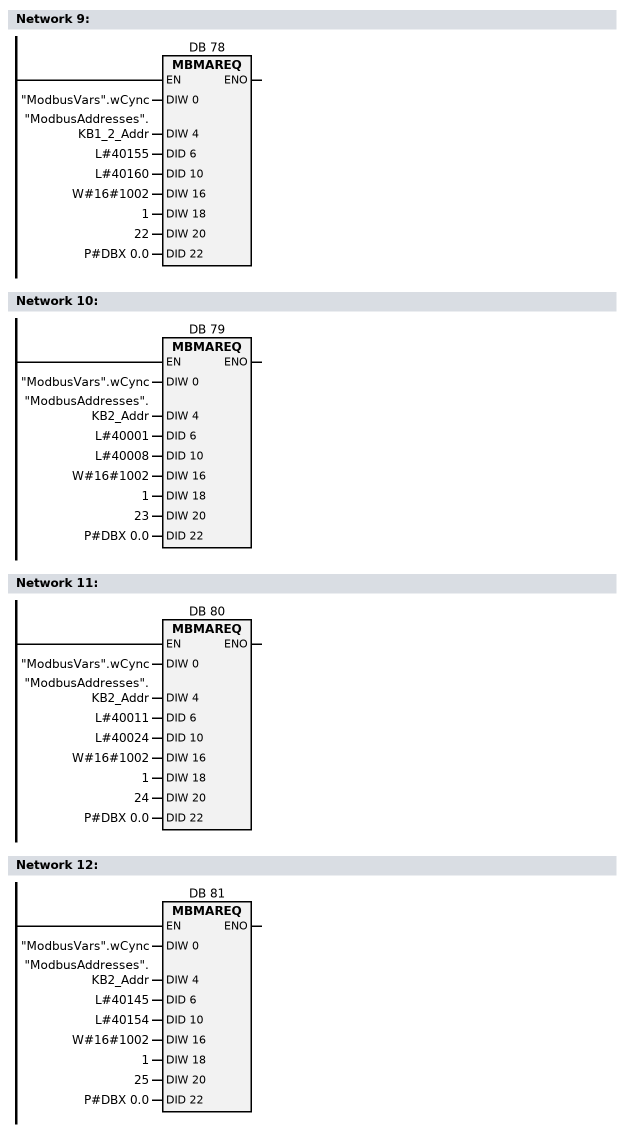
NETWORK
TITLE =
      CALL  "MBMAREQ" , DB 78 (
           DIW 0                    := "ModbusVars".wCync,
           DIW 4                    := "ModbusAddresses".KB1_2_Addr,
           DID 6                    := L#40155,
           DID 10                   := L#40160,
           DIW 16                   := W#16#1002,
           DIW 18                   := 1,
           DIW 20                   := 22,
           DID 22                   := P#DBX 0.0);
      NOP   0;
NETWORK
TITLE =
      CALL  "MBMAREQ" , DB 79 (
           DIW 0                    := "ModbusVars".wCync,
           DIW 4                    := "ModbusAddresses".KB2_Addr,
           DID 6                    := L#40001,
           DID 10                   := L#40008,
           DIW 16                   := W#16#1002,
           DIW 18                   := 1,
           DIW 20                   := 23,
           DID 22                   := P#DBX 0.0);
      NOP   0;
NETWORK
TITLE =
      CALL  "MBMAREQ" , DB 80 (
           DIW 0                    := "ModbusVars".wCync,
           DIW 4                    := "ModbusAddresses".KB2_Addr,
           DID 6                    := L#40011,
           DID 10                   := L#40024,
           DIW 16                   := W#16#1002,
           DIW 18                   := 1,
           DIW 20                   := 24,
           DID 22                   := P#DBX 0.0);
      NOP   0;
NETWORK
TITLE =
      CALL  "MBMAREQ" , DB 81 (
           DIW 0                    := "ModbusVars".wCync,
           DIW 4                    := "ModbusAddresses".KB2_Addr,
           DID 6                    := L#40145,
           DID 10                   := L#40154,
           DIW 16                   := W#16#1002,
           DIW 18                   := 1,
           DIW 20                   := 25,
           DID 22                   := P#DBX 0.0);
      NOP   0;
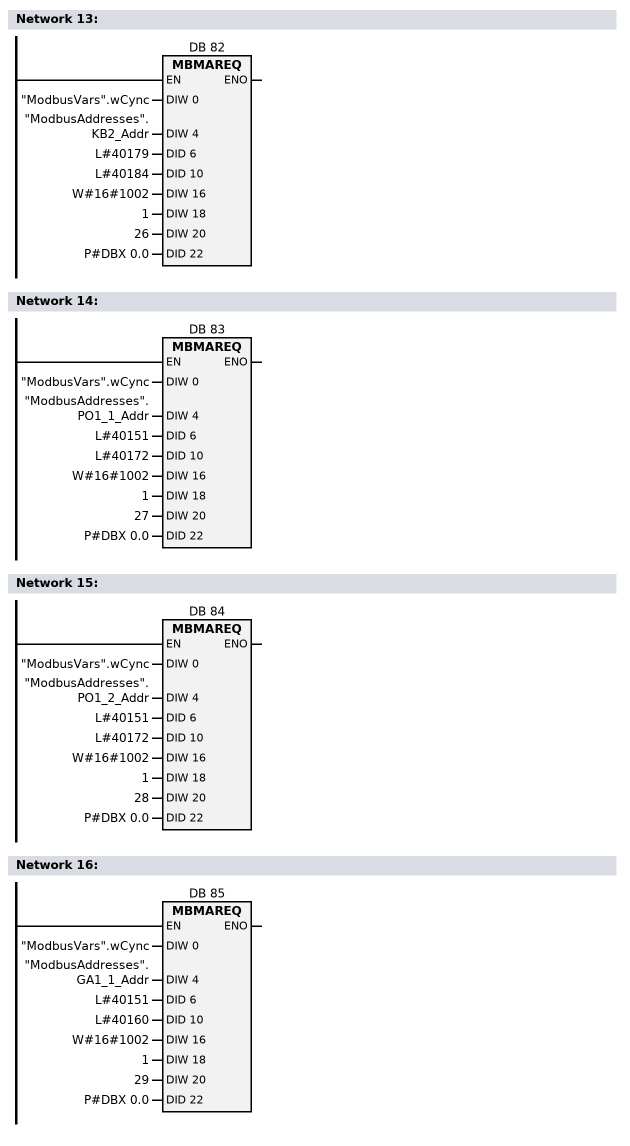
NETWORK
TITLE =
      CALL  "MBMAREQ" , DB 82 (
           DIW 0                    := "ModbusVars".wCync,
           DIW 4                    := "ModbusAddresses".KB2_Addr,
           DID 6                    := L#40179,
           DID 10                   := L#40184,
           DIW 16                   := W#16#1002,
           DIW 18                   := 1,
           DIW 20                   := 26,
           DID 22                   := P#DBX 0.0);
      NOP   0;
NETWORK
TITLE =
      CALL  "MBMAREQ" , DB 83 (
           DIW 0                    := "ModbusVars".wCync,
           DIW 4                    := "ModbusAddresses".PO1_1_Addr,
           DID 6                    := L#40151,
           DID 10                   := L#40172,
           DIW 16                   := W#16#1002,
           DIW 18                   := 1,
           DIW 20                   := 27,
           DID 22                   := P#DBX 0.0);
      NOP   0;
NETWORK
TITLE =
      CALL  "MBMAREQ" , DB 84 (
           DIW 0                    := "ModbusVars".wCync,
           DIW 4                    := "ModbusAddresses".PO1_2_Addr,
           DID 6                    := L#40151,
           DID 10                   := L#40172,
           DIW 16                   := W#16#1002,
           DIW 18                   := 1,
           DIW 20                   := 28,
           DID 22                   := P#DBX 0.0);
      NOP   0;
NETWORK
TITLE =
      CALL  "MBMAREQ" , DB 85 (
           DIW 0                    := "ModbusVars".wCync,
           DIW 4                    := "ModbusAddresses".GA1_1_Addr,
           DID 6                    := L#40151,
           DID 10                   := L#40160,
           DIW 16                   := W#16#1002,
           DIW 18                   := 1,
           DIW 20                   := 29,
           DID 22                   := P#DBX 0.0);
      NOP   0;
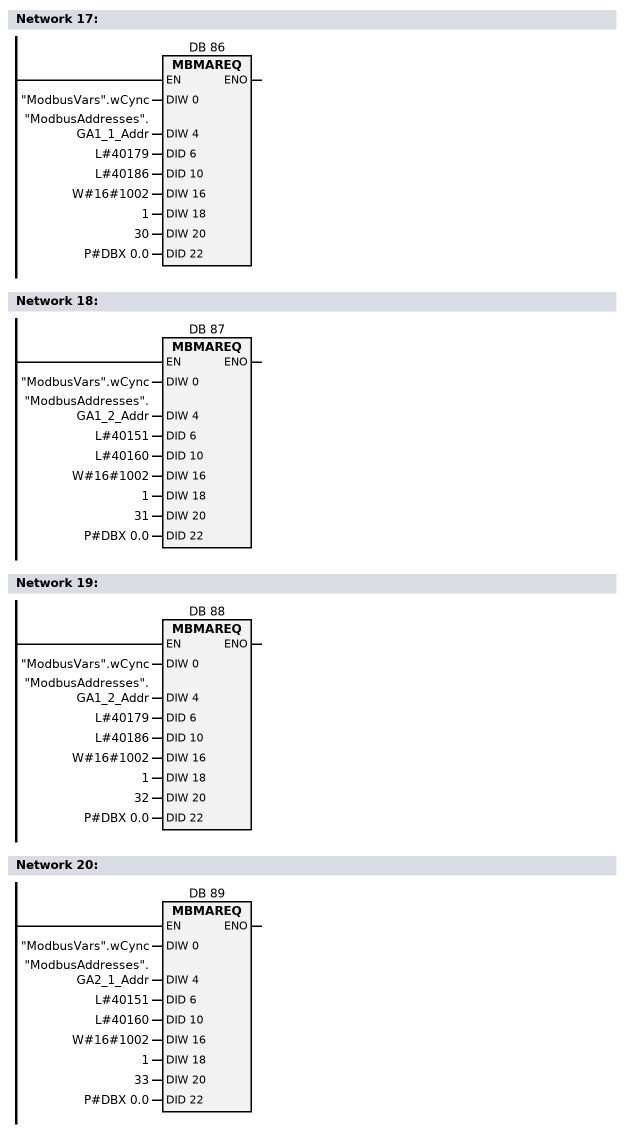
NETWORK
TITLE =
      CALL  "MBMAREQ" , DB 86 (
           DIW 0                    := "ModbusVars".wCync,
           DIW 4                    := "ModbusAddresses".GA1_1_Addr,
           DID 6                    := L#40179,
           DID 10                   := L#40186,
           DIW 16                   := W#16#1002,
           DIW 18                   := 1,
           DIW 20                   := 30,
           DID 22                   := P#DBX 0.0);
      NOP   0;
NETWORK
TITLE =
      CALL  "MBMAREQ" , DB 87 (
           DIW 0                    := "ModbusVars".wCync,
           DIW 4                    := "ModbusAddresses".GA1_2_Addr,
           DID 6                    := L#40151,
           DID 10                   := L#40160,
           DIW 16                   := W#16#1002,
           DIW 18                   := 1,
           DIW 20                   := 31,
           DID 22                   := P#DBX 0.0);
      NOP   0;
NETWORK
TITLE =
      CALL  "MBMAREQ" , DB 88 (
           DIW 0                    := "ModbusVars".wCync,
           DIW 4                    := "ModbusAddresses".GA1_2_Addr,
           DID 6                    := L#40179,
           DID 10                   := L#40186,
           DIW 16                   := W#16#1002,
           DIW 18                   := 1,
           DIW 20                   := 32,
           DID 22                   := P#DBX 0.0);
      NOP   0;
NETWORK
TITLE =
      CALL  "MBMAREQ" , DB 89 (
           DIW 0                    := "ModbusVars".wCync,
           DIW 4                    := "ModbusAddresses".GA2_1_Addr,
           DID 6                    := L#40151,
           DID 10                   := L#40160,
           DIW 16                   := W#16#1002,
           DIW 18                   := 1,
           DIW 20                   := 33,
           DID 22                   := P#DBX 0.0);
      NOP   0;
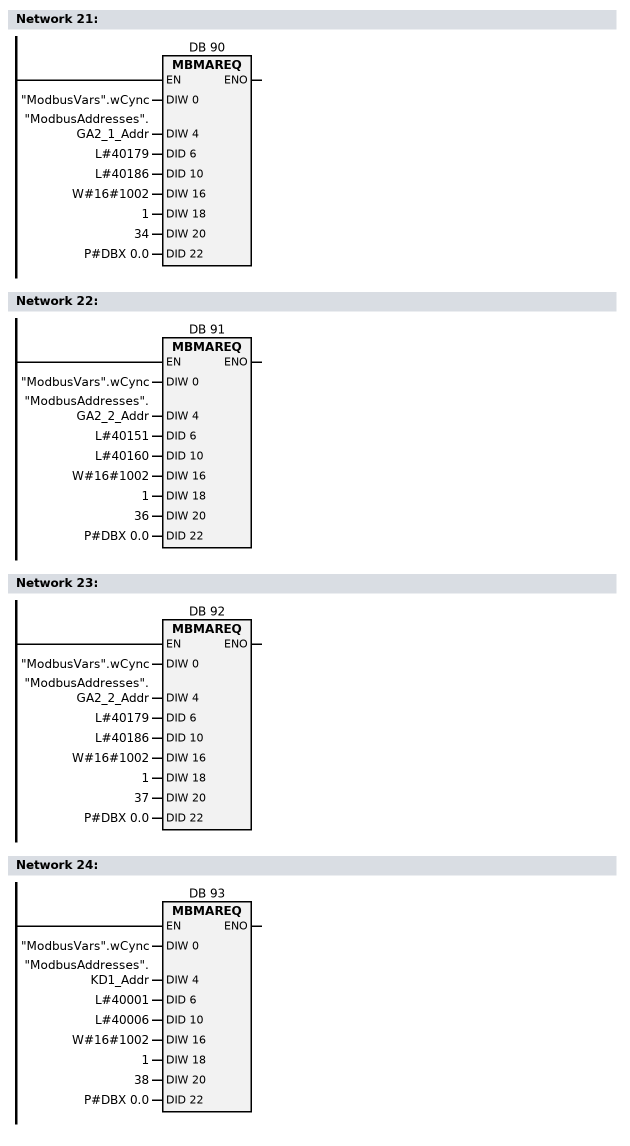
NETWORK
TITLE =
      CALL  "MBMAREQ" , DB 90 (
           DIW 0                    := "ModbusVars".wCync,
           DIW 4                    := "ModbusAddresses".GA2_1_Addr,
           DID 6                    := L#40179,
           DID 10                   := L#40186,
           DIW 16                   := W#16#1002,
           DIW 18                   := 1,
           DIW 20                   := 34,
           DID 22                   := P#DBX 0.0);
      NOP   0;
NETWORK
TITLE =
      CALL  "MBMAREQ" , DB 91 (
           DIW 0                    := "ModbusVars".wCync,
           DIW 4                    := "ModbusAddresses".GA2_2_Addr,
           DID 6                    := L#40151,
           DID 10                   := L#40160,
           DIW 16                   := W#16#1002,
           DIW 18                   := 1,
           DIW 20                   := 36,
           DID 22                   := P#DBX 0.0);
      NOP   0;
NETWORK
TITLE =
      CALL  "MBMAREQ" , DB 92 (
           DIW 0                    := "ModbusVars".wCync,
           DIW 4                    := "ModbusAddresses".GA2_2_Addr,
           DID 6                    := L#40179,
           DID 10                   := L#40186,
           DIW 16                   := W#16#1002,
           DIW 18                   := 1,
           DIW 20                   := 37,
           DID 22                   := P#DBX 0.0);
      NOP   0;
NETWORK
TITLE =
      CALL  "MBMAREQ" , DB 93 (
           DIW 0                    := "ModbusVars".wCync,
           DIW 4                    := "ModbusAddresses".KD1_Addr,
           DID 6                    := L#40001,
           DID 10                   := L#40006,
           DIW 16                   := W#16#1002,
           DIW 18                   := 1,
           DIW 20                   := 38,
           DID 22                   := P#DBX 0.0);
      NOP   0;
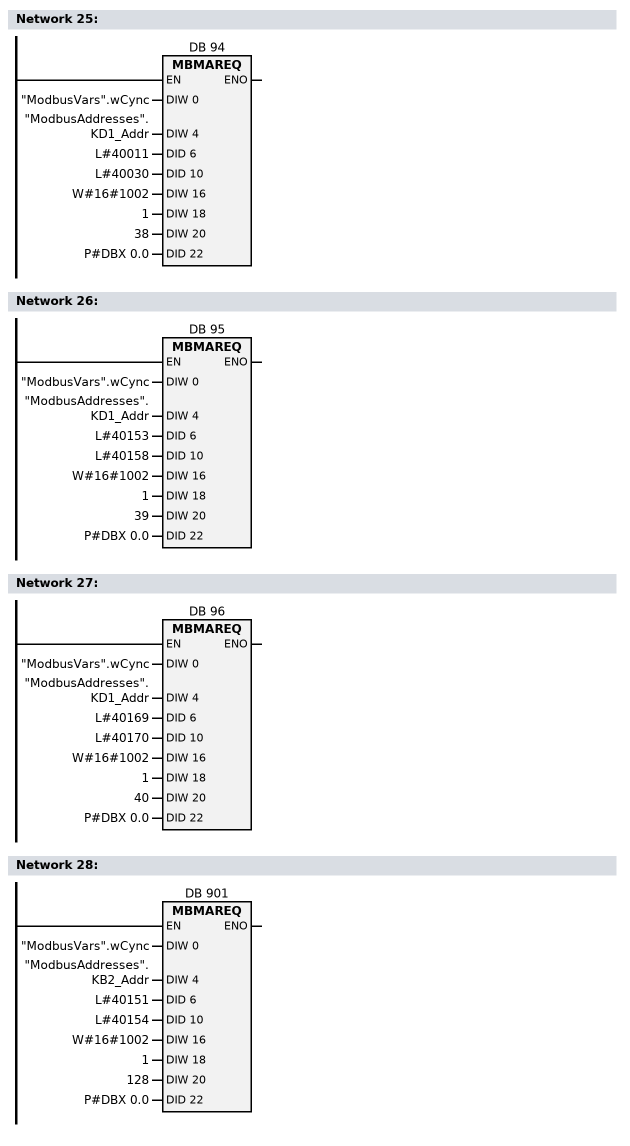
NETWORK
TITLE =
      CALL  "MBMAREQ" , DB 94 (
           DIW 0                    := "ModbusVars".wCync,
           DIW 4                    := "ModbusAddresses".KD1_Addr,
           DID 6                    := L#40011,
           DID 10                   := L#40030,
           DIW 16                   := W#16#1002,
           DIW 18                   := 1,
           DIW 20                   := 38,
           DID 22                   := P#DBX 0.0);
      NOP   0;
NETWORK
TITLE =
      CALL  "MBMAREQ" , DB 95 (
           DIW 0                    := "ModbusVars".wCync,
           DIW 4                    := "ModbusAddresses".KD1_Addr,
           DID 6                    := L#40153,
           DID 10                   := L#40158,
           DIW 16                   := W#16#1002,
           DIW 18                   := 1,
           DIW 20                   := 39,
           DID 22                   := P#DBX 0.0);
      NOP   0;
NETWORK
TITLE =
      CALL  "MBMAREQ" , DB 96 (
           DIW 0                    := "ModbusVars".wCync,
           DIW 4                    := "ModbusAddresses".KD1_Addr,
           DID 6                    := L#40169,
           DID 10                   := L#40170,
           DIW 16                   := W#16#1002,
           DIW 18                   := 1,
           DIW 20                   := 40,
           DID 22                   := P#DBX 0.0);
      NOP   0;
NETWORK
TITLE =
      CALL  "MBMAREQ" , DB 901 (
           DIW 0                    := "ModbusVars".wCync,
           DIW 4                    := "ModbusAddresses".KB2_Addr,
           DID 6                    := L#40151,
           DID 10                   := L#40154,
           DIW 16                   := W#16#1002,
           DIW 18                   := 1,
           DIW 20                   := 128,
           DID 22                   := P#DBX 0.0);
      NOP   0;
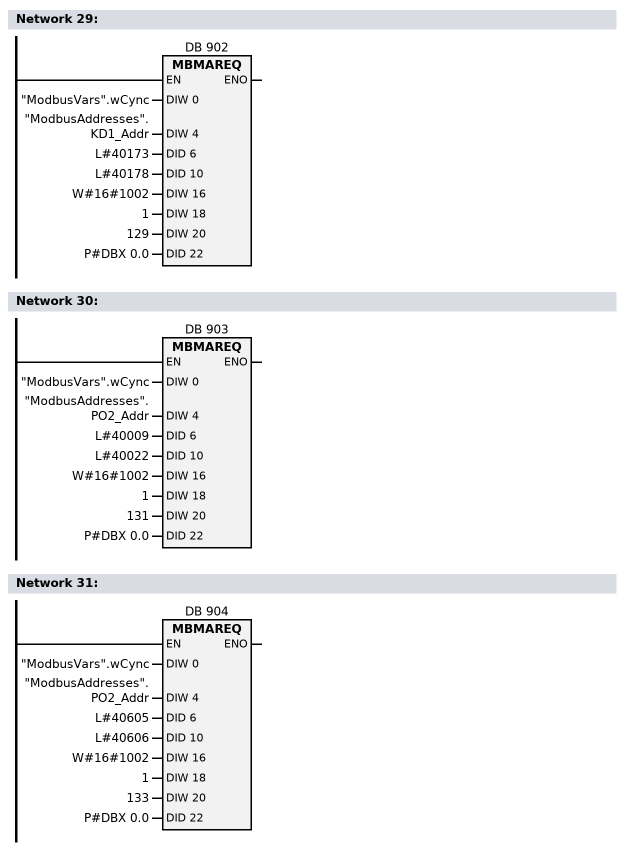
NETWORK
TITLE =
      CALL  "MBMAREQ" , DB 902 (
           DIW 0                    := "ModbusVars".wCync,
           DIW 4                    := "ModbusAddresses".KD1_Addr,
           DID 6                    := L#40173,
           DID 10                   := L#40178,
           DIW 16                   := W#16#1002,
           DIW 18                   := 1,
           DIW 20                   := 129,
           DID 22                   := P#DBX 0.0);
      NOP   0;
NETWORK
TITLE =
      CALL  "MBMAREQ" , DB 903 (
           DIW 0                    := "ModbusVars".wCync,
           DIW 4                    := "ModbusAddresses".PO2_Addr,
           DID 6                    := L#40009,
           DID 10                   := L#40022,
           DIW 16                   := W#16#1002,
           DIW 18                   := 1,
           DIW 20                   := 131,
           DID 22                   := P#DBX 0.0);
      NOP   0;
NETWORK
TITLE =
      CALL  "MBMAREQ" , DB 904 (
           DIW 0                    := "ModbusVars".wCync,
           DIW 4                    := "ModbusAddresses".PO2_Addr,
           DID 6                    := L#40605,
           DID 10                   := L#40606,
           DIW 16                   := W#16#1002,
           DIW 18                   := 1,
           DIW 20                   := 133,
           DID 22                   := P#DBX 0.0);
      NOP   0;
END_FUNCTION_BLOCK

FUNCTION_BLOCK "ModbusCoils"	// FB 16
VERSION : 0.1
BEGIN
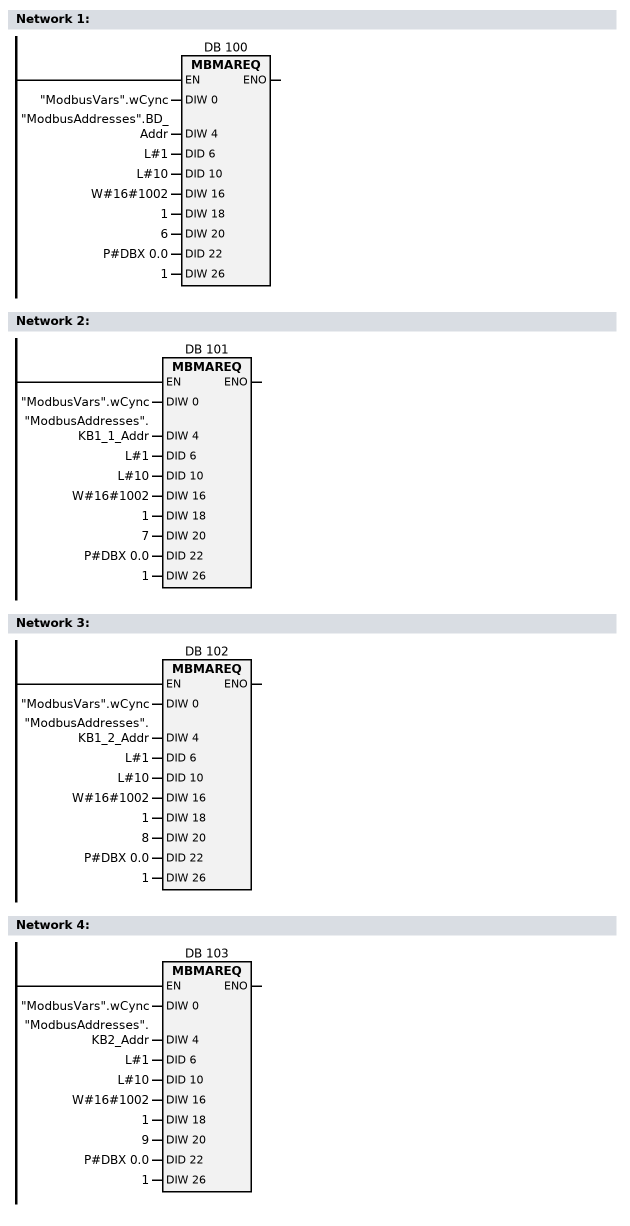
NETWORK
TITLE =
      CALL  "MBMAREQ" , DB 100 (
           DIW 0                    := "ModbusVars".wCync,
           DIW 4                    := "ModbusAddresses".BD_Addr,
           DID 6                    := L#1,
           DID 10                   := L#10,
           DIW 16                   := W#16#1002,
           DIW 18                   := 1,
           DIW 20                   := 6,
           DID 22                   := P#DBX 0.0,
           DIW 26                   := 1);
      NOP   0;
NETWORK
TITLE =
      CALL  "MBMAREQ" , DB 101 (
           DIW 0                    := "ModbusVars".wCync,
           DIW 4                    := "ModbusAddresses".KB1_1_Addr,
           DID 6                    := L#1,
           DID 10                   := L#10,
           DIW 16                   := W#16#1002,
           DIW 18                   := 1,
           DIW 20                   := 7,
           DID 22                   := P#DBX 0.0,
           DIW 26                   := 1);
      NOP   0;
NETWORK
TITLE =
      CALL  "MBMAREQ" , DB 102 (
           DIW 0                    := "ModbusVars".wCync,
           DIW 4                    := "ModbusAddresses".KB1_2_Addr,
           DID 6                    := L#1,
           DID 10                   := L#10,
           DIW 16                   := W#16#1002,
           DIW 18                   := 1,
           DIW 20                   := 8,
           DID 22                   := P#DBX 0.0,
           DIW 26                   := 1);
      NOP   0;
NETWORK
TITLE =
      CALL  "MBMAREQ" , DB 103 (
           DIW 0                    := "ModbusVars".wCync,
           DIW 4                    := "ModbusAddresses".KB2_Addr,
           DID 6                    := L#1,
           DID 10                   := L#10,
           DIW 16                   := W#16#1002,
           DIW 18                   := 1,
           DIW 20                   := 9,
           DID 22                   := P#DBX 0.0,
           DIW 26                   := 1);
      NOP   0;
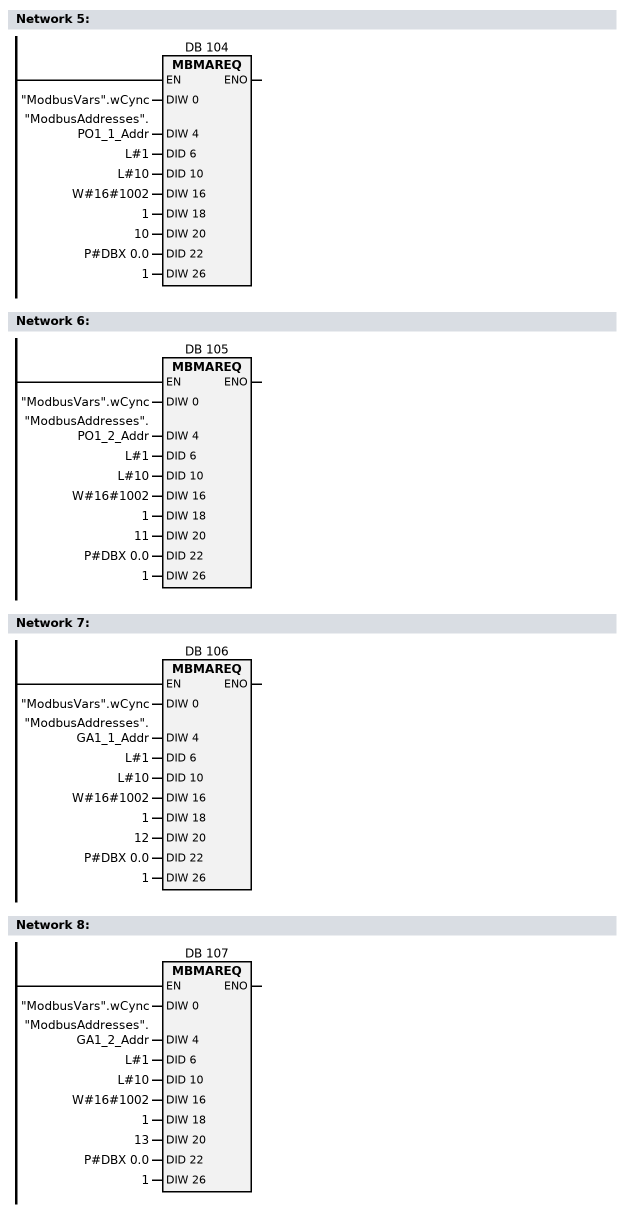
NETWORK
TITLE =
      CALL  "MBMAREQ" , DB 104 (
           DIW 0                    := "ModbusVars".wCync,
           DIW 4                    := "ModbusAddresses".PO1_1_Addr,
           DID 6                    := L#1,
           DID 10                   := L#10,
           DIW 16                   := W#16#1002,
           DIW 18                   := 1,
           DIW 20                   := 10,
           DID 22                   := P#DBX 0.0,
           DIW 26                   := 1);
      NOP   0;
NETWORK
TITLE =
      CALL  "MBMAREQ" , DB 105 (
           DIW 0                    := "ModbusVars".wCync,
           DIW 4                    := "ModbusAddresses".PO1_2_Addr,
           DID 6                    := L#1,
           DID 10                   := L#10,
           DIW 16                   := W#16#1002,
           DIW 18                   := 1,
           DIW 20                   := 11,
           DID 22                   := P#DBX 0.0,
           DIW 26                   := 1);
      NOP   0;
NETWORK
TITLE =
      CALL  "MBMAREQ" , DB 106 (
           DIW 0                    := "ModbusVars".wCync,
           DIW 4                    := "ModbusAddresses".GA1_1_Addr,
           DID 6                    := L#1,
           DID 10                   := L#10,
           DIW 16                   := W#16#1002,
           DIW 18                   := 1,
           DIW 20                   := 12,
           DID 22                   := P#DBX 0.0,
           DIW 26                   := 1);
      NOP   0;
NETWORK
TITLE =
      CALL  "MBMAREQ" , DB 107 (
           DIW 0                    := "ModbusVars".wCync,
           DIW 4                    := "ModbusAddresses".GA1_2_Addr,
           DID 6                    := L#1,
           DID 10                   := L#10,
           DIW 16                   := W#16#1002,
           DIW 18                   := 1,
           DIW 20                   := 13,
           DID 22                   := P#DBX 0.0,
           DIW 26                   := 1);
      NOP   0;
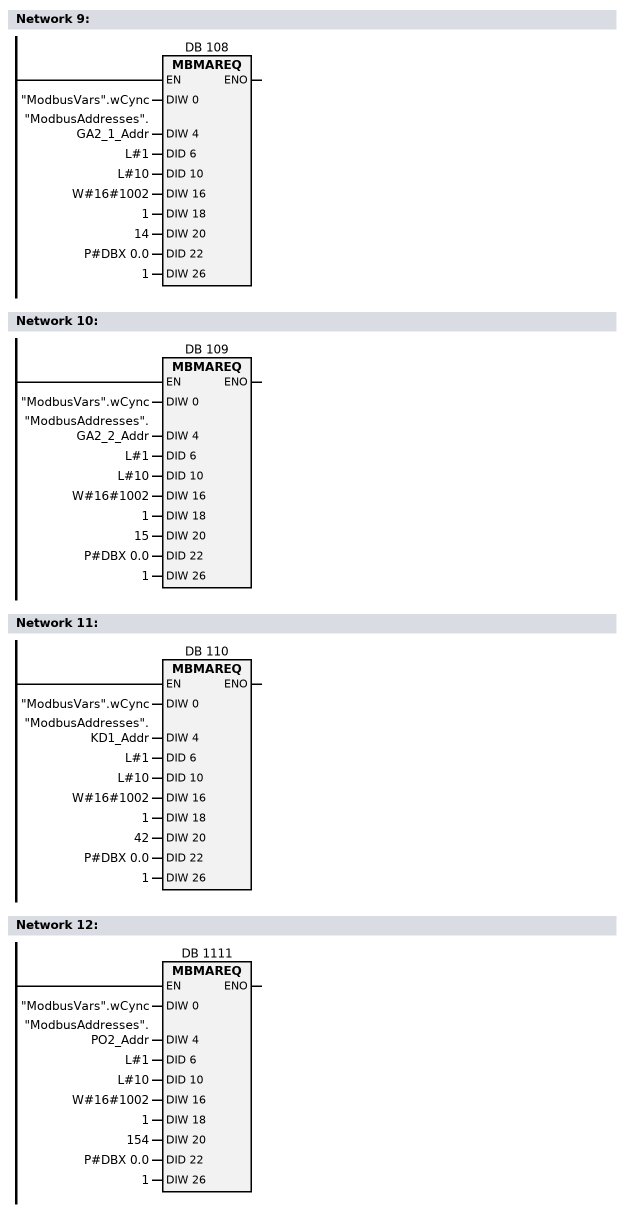
NETWORK
TITLE =
      CALL  "MBMAREQ" , DB 108 (
           DIW 0                    := "ModbusVars".wCync,
           DIW 4                    := "ModbusAddresses".GA2_1_Addr,
           DID 6                    := L#1,
           DID 10                   := L#10,
           DIW 16                   := W#16#1002,
           DIW 18                   := 1,
           DIW 20                   := 14,
           DID 22                   := P#DBX 0.0,
           DIW 26                   := 1);
      NOP   0;
NETWORK
TITLE =
      CALL  "MBMAREQ" , DB 109 (
           DIW 0                    := "ModbusVars".wCync,
           DIW 4                    := "ModbusAddresses".GA2_2_Addr,
           DID 6                    := L#1,
           DID 10                   := L#10,
           DIW 16                   := W#16#1002,
           DIW 18                   := 1,
           DIW 20                   := 15,
           DID 22                   := P#DBX 0.0,
           DIW 26                   := 1);
      NOP   0;
NETWORK
TITLE =
      CALL  "MBMAREQ" , DB 110 (
           DIW 0                    := "ModbusVars".wCync,
           DIW 4                    := "ModbusAddresses".KD1_Addr,
           DID 6                    := L#1,
           DID 10                   := L#10,
           DIW 16                   := W#16#1002,
           DIW 18                   := 1,
           DIW 20                   := 42,
           DID 22                   := P#DBX 0.0,
           DIW 26                   := 1);
      NOP   0;
NETWORK
TITLE =
      CALL  "MBMAREQ" , DB 1111 (
           DIW 0                    := "ModbusVars".wCync,
           DIW 4                    := "ModbusAddresses".PO2_Addr,
           DID 6                    := L#1,
           DID 10                   := L#10,
           DIW 16                   := W#16#1002,
           DIW 18                   := 1,
           DIW 20                   := 154,
           DID 22                   := P#DBX 0.0,
           DIW 26                   := 1);
      NOP   0;
END_FUNCTION_BLOCK

FUNCTION_BLOCK "ModbusOutputs"	// FB 17
VERSION : 0.1
BEGIN
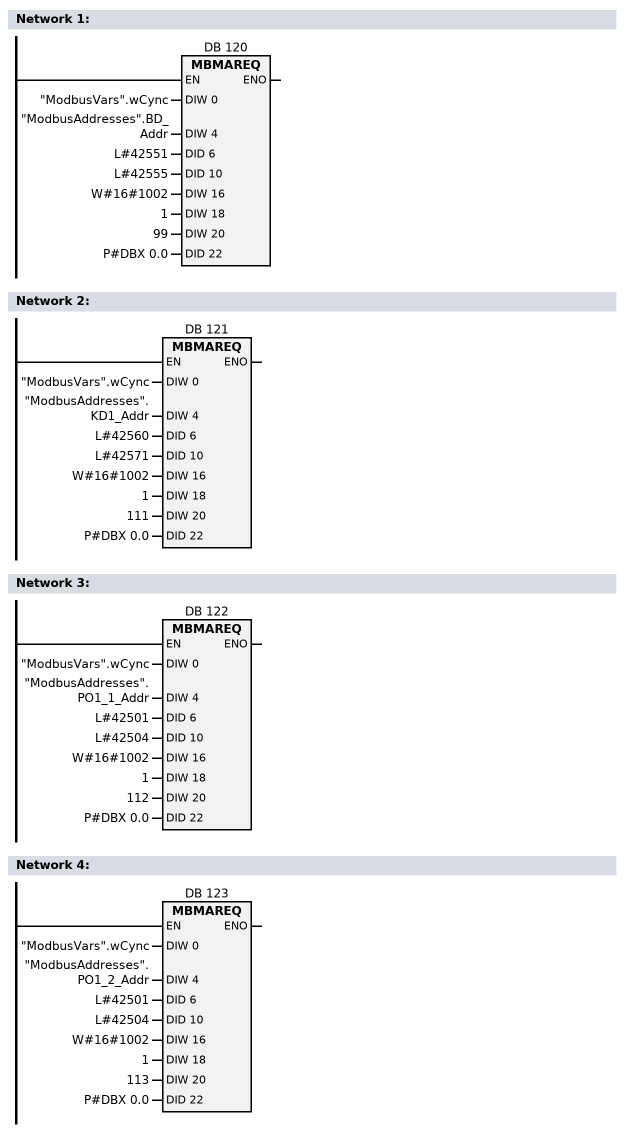
NETWORK
TITLE =
      CALL  "MBMAREQ" , DB 120 (
           DIW 0                    := "ModbusVars".wCync,
           DIW 4                    := "ModbusAddresses".BD_Addr,
           DID 6                    := L#42551,
           DID 10                   := L#42555,
           DIW 16                   := W#16#1002,
           DIW 18                   := 1,
           DIW 20                   := 99,
           DID 22                   := P#DBX 0.0);
      NOP   0;
NETWORK
TITLE =
      CALL  "MBMAREQ" , DB 121 (
           DIW 0                    := "ModbusVars".wCync,
           DIW 4                    := "ModbusAddresses".KD1_Addr,
           DID 6                    := L#42560,
           DID 10                   := L#42571,
           DIW 16                   := W#16#1002,
           DIW 18                   := 1,
           DIW 20                   := 111,
           DID 22                   := P#DBX 0.0);
      NOP   0;
NETWORK
TITLE =
      CALL  "MBMAREQ" , DB 122 (
           DIW 0                    := "ModbusVars".wCync,
           DIW 4                    := "ModbusAddresses".PO1_1_Addr,
           DID 6                    := L#42501,
           DID 10                   := L#42504,
           DIW 16                   := W#16#1002,
           DIW 18                   := 1,
           DIW 20                   := 112,
           DID 22                   := P#DBX 0.0);
      NOP   0;
NETWORK
TITLE =
      CALL  "MBMAREQ" , DB 123 (
           DIW 0                    := "ModbusVars".wCync,
           DIW 4                    := "ModbusAddresses".PO1_2_Addr,
           DID 6                    := L#42501,
           DID 10                   := L#42504,
           DIW 16                   := W#16#1002,
           DIW 18                   := 1,
           DIW 20                   := 113,
           DID 22                   := P#DBX 0.0);
      NOP   0;
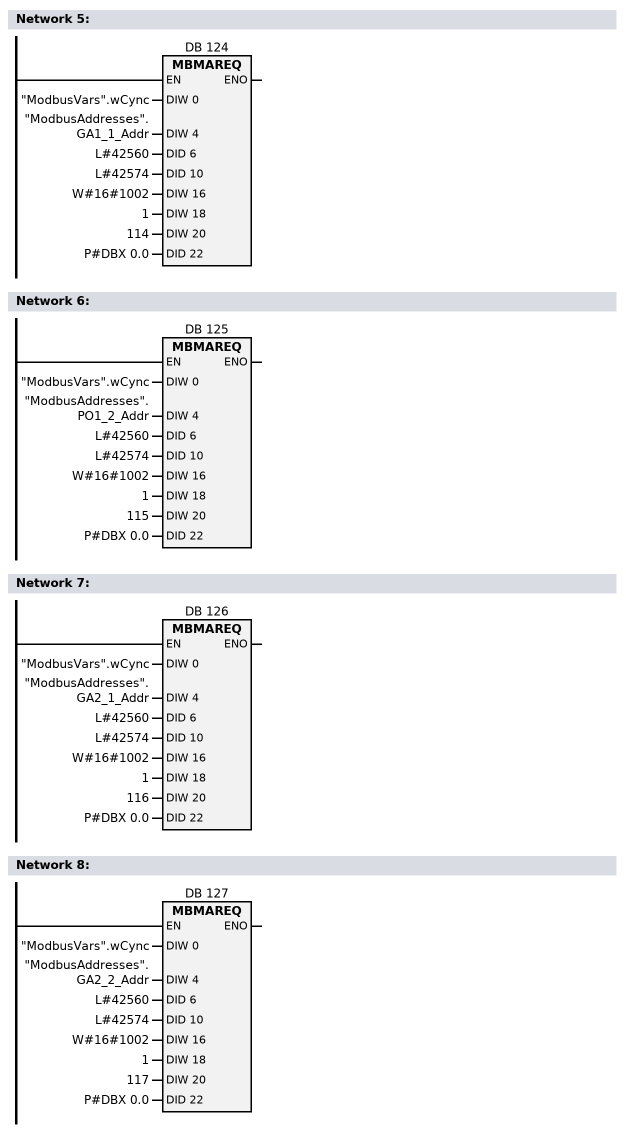
NETWORK
TITLE =
      CALL  "MBMAREQ" , DB 124 (
           DIW 0                    := "ModbusVars".wCync,
           DIW 4                    := "ModbusAddresses".GA1_1_Addr,
           DID 6                    := L#42560,
           DID 10                   := L#42574,
           DIW 16                   := W#16#1002,
           DIW 18                   := 1,
           DIW 20                   := 114,
           DID 22                   := P#DBX 0.0);
      NOP   0;
NETWORK
TITLE =
      CALL  "MBMAREQ" , DB 125 (
           DIW 0                    := "ModbusVars".wCync,
           DIW 4                    := "ModbusAddresses".PO1_2_Addr,
           DID 6                    := L#42560,
           DID 10                   := L#42574,
           DIW 16                   := W#16#1002,
           DIW 18                   := 1,
           DIW 20                   := 115,
           DID 22                   := P#DBX 0.0);
      NOP   0;
NETWORK
TITLE =
      CALL  "MBMAREQ" , DB 126 (
           DIW 0                    := "ModbusVars".wCync,
           DIW 4                    := "ModbusAddresses".GA2_1_Addr,
           DID 6                    := L#42560,
           DID 10                   := L#42574,
           DIW 16                   := W#16#1002,
           DIW 18                   := 1,
           DIW 20                   := 116,
           DID 22                   := P#DBX 0.0);
      NOP   0;
NETWORK
TITLE =
      CALL  "MBMAREQ" , DB 127 (
           DIW 0                    := "ModbusVars".wCync,
           DIW 4                    := "ModbusAddresses".GA2_2_Addr,
           DID 6                    := L#42560,
           DID 10                   := L#42574,
           DIW 16                   := W#16#1002,
           DIW 18                   := 1,
           DIW 20                   := 117,
           DID 22                   := P#DBX 0.0);
      NOP   0;
END_FUNCTION_BLOCK

FUNCTION_BLOCK "BD_GetOutputs"	// FB 18
VERSION : 0.1
BEGIN
NETWORK
TITLE =
      CALL  "fnWordPack" (
           bHigh                    := "BD_OutputBytes_1".arBytes[0],
           bLow                     := "BD_OutputBytes_1".arBytes[1],
           OUT                      := "BD_Outputs_1".DryerMotor);
NETWORK
TITLE =
      CALL  "fnWordPack" (
           bHigh                    := "BD_OutputBytes_1".arBytes[2],
           bLow                     := "BD_OutputBytes_1".arBytes[3],
           OUT                      := "BD_Outputs_1".PDPAlarm);
NETWORK
TITLE =
      CALL  "fnWordPack" (
           bHigh                    := "BD_OutputBytes_1".arBytes[4],
           bLow                     := "BD_OutputBytes_1".arBytes[5],
           OUT                      := "BD_Outputs_1".GeneralShutdown);
NETWORK
TITLE =
      CALL  "fnWordPack" (
           bHigh                    := "BD_OutputBytes_1".arBytes[6],
           bLow                     := "BD_OutputBytes_1".arBytes[7],
           OUT                      := "BD_Outputs_1".GeneralWarning);
NETWORK
TITLE =
      CALL  "fnWordPack" (
           bHigh                    := "BD_OutputBytes_1".arBytes[8],
           bLow                     := "BD_OutputBytes_1".arBytes[9],
           OUT                      := "BD_Outputs_1".LowPressureAlarm);
NETWORK
TITLE =
      CALL  "fnWordPack" (
           bHigh                    := "BD_OutputBytes_2".arBytes[0],
           bLow                     := "BD_OutputBytes_2".arBytes[1],
           OUT                      := "BD_Outputs_2".BlowerContactor);
NETWORK
TITLE =
      CALL  "fnWordPack" (
           bHigh                    := "BD_OutputBytes_2".arBytes[2],
           bLow                     := "BD_OutputBytes_2".arBytes[3],
           OUT                      := "BD_Outputs_2".MainHeaters);
NETWORK
TITLE =
      CALL  "fnWordPack" (
           bHigh                    := "BD_OutputBytes_2".arBytes[4],
           bLow                     := "BD_OutputBytes_2".arBytes[5],
           OUT                      := "BD_Outputs_2".RegulatingHeaters);
NETWORK
TITLE =
      CALL  "fnWordPack" (
           bHigh                    := "BD_OutputBytes_2".arBytes[6],
           bLow                     := "BD_OutputBytes_2".arBytes[7],
           OUT                      := "BD_Outputs_2".ValveV1Opened);
NETWORK
TITLE =
      CALL  "fnWordPack" (
           bHigh                    := "BD_OutputBytes_2".arBytes[8],
           bLow                     := "BD_OutputBytes_2".arBytes[9],
           OUT                      := "BD_Outputs_2".ValveV1Closed);
NETWORK
TITLE =
      CALL  "fnWordPack" (
           bHigh                    := "BD_OutputBytes_2".arBytes[10],
           bLow                     := "BD_OutputBytes_2".arBytes[11],
           OUT                      := "BD_Outputs_2".ValveV2Opened);
NETWORK
TITLE =
      CALL  "fnWordPack" (
           bHigh                    := "BD_OutputBytes_2".arBytes[12],
           bLow                     := "BD_OutputBytes_2".arBytes[13],
           OUT                      := "BD_Outputs_2".ValveV2Closed);
NETWORK
TITLE =
      CALL  "fnWordPack" (
           bHigh                    := "BD_OutputBytes_2".arBytes[14],
           bLow                     := "BD_OutputBytes_2".arBytes[15],
           OUT                      := "BD_Outputs_2".RegValveVesselA);
NETWORK
TITLE =
      CALL  "fnWordPack" (
           bHigh                    := "BD_OutputBytes_2".arBytes[16],
           bLow                     := "BD_OutputBytes_2".arBytes[17],
           OUT                      := "BD_Outputs_2".RegValveVesselB);
NETWORK
TITLE =
      CALL  "fnWordPack" (
           bHigh                    := "BD_OutputBytes_2".arBytes[18],
           bLow                     := "BD_OutputBytes_2".arBytes[19],
           OUT                      := "BD_Outputs_2".CoolingAirValveAOpen);
NETWORK
TITLE =
      CALL  "fnWordPack" (
           bHigh                    := "BD_OutputBytes_2".arBytes[20],
           bLow                     := "BD_OutputBytes_2".arBytes[21],
           OUT                      := "BD_Outputs_2".CoolingAirValveBOpen);
NETWORK
TITLE =
      CALL  "fnWordPack" (
           bHigh                    := "BD_OutputBytes_2".arBytes[22],
           bLow                     := "BD_OutputBytes_2".arBytes[23],
           OUT                      := "BD_Outputs_2".PressureReliefValveA);
NETWORK
TITLE =
      CALL  "fnWordPack" (
           bHigh                    := "BD_OutputBytes_2".arBytes[24],
           bLow                     := "BD_OutputBytes_2".arBytes[25],
           OUT                      := "BD_Outputs_2".PressureReliefValvegB);
END_FUNCTION_BLOCK

FUNCTION_BLOCK "PO1_1_GetOutputs"	// FB 19
VERSION : 0.1
BEGIN
NETWORK
TITLE =
      CALL  "fnBytesToRealTwoComas" (
           bHigh                    := "PO1_1_OutBytes".arBytes[0],
           bLow                     := "PO1_1_OutBytes".arBytes[1],
           OUT                      := "PO1_1_Outputs".EEV1);
NETWORK
TITLE =
      CALL  "fnBytesToRealTwoComas" (
           bHigh                    := "PO1_1_OutBytes".arBytes[2],
           bLow                     := "PO1_1_OutBytes".arBytes[3],
           OUT                      := "PO1_1_Outputs".EEV2);
NETWORK
TITLE =
      CALL  "fnBytesToRealTwoComas" (
           bHigh                    := "PO1_1_OutBytes".arBytes[4],
           bLow                     := "PO1_1_OutBytes".arBytes[5],
           OUT                      := "PO1_1_Outputs".HGBP1);
NETWORK
TITLE =
      CALL  "fnBytesToRealTwoComas" (
           bHigh                    := "PO1_1_OutBytes".arBytes[6],
           bLow                     := "PO1_1_OutBytes".arBytes[7],
           OUT                      := "PO1_1_Outputs".HGBP2);
END_FUNCTION_BLOCK

FUNCTION_BLOCK "PO1_2_GetOutputs"	// FB 20
VERSION : 0.1
BEGIN
NETWORK
TITLE =
      CALL  "fnBytesToRealTwoComas" (
           bHigh                    := "PO1_2_OutBytes".arBytes[0],
           bLow                     := "PO1_2_OutBytes".arBytes[1],
           OUT                      := "PO1_2_Outputs".EEV1);
NETWORK
TITLE =
      CALL  "fnBytesToRealTwoComas" (
           bHigh                    := "PO1_2_OutBytes".arBytes[2],
           bLow                     := "PO1_2_OutBytes".arBytes[3],
           OUT                      := "PO1_2_Outputs".EEV2);
NETWORK
TITLE =
      CALL  "fnBytesToRealTwoComas" (
           bHigh                    := "PO1_2_OutBytes".arBytes[4],
           bLow                     := "PO1_2_OutBytes".arBytes[5],
           OUT                      := "PO1_2_Outputs".HGBP1);
NETWORK
TITLE =
      CALL  "fnBytesToRealTwoComas" (
           bHigh                    := "PO1_2_OutBytes".arBytes[6],
           bLow                     := "PO1_2_OutBytes".arBytes[7],
           OUT                      := "PO1_2_Outputs".HGBP2);
END_FUNCTION_BLOCK

FUNCTION_BLOCK "GA1_1_GetOutputs"	// FB 21
VERSION : 0.1
BEGIN
NETWORK
TITLE =
      CALL  "fnWordPack" (
           bHigh                    := "GA1_1_OutBytes".arBytes[0],
           bLow                     := "GA1_1_OutBytes".arBytes[1],
           OUT                      := "GA1_1_Outputs".InletValveVesselA);
NETWORK
TITLE =
      CALL  "fnWordPack" (
           bHigh                    := "GA1_1_OutBytes".arBytes[2],
           bLow                     := "GA1_1_OutBytes".arBytes[3],
           OUT                      := "GA1_1_Outputs".InletValveVesselB);
NETWORK
TITLE =
      CALL  "fnWordPack" (
           bHigh                    := "GA1_1_OutBytes".arBytes[4],
           bLow                     := "GA1_1_OutBytes".arBytes[5],
           OUT                      := "GA1_1_Outputs".EqualizationValve);
NETWORK
TITLE =
      CALL  "fnWordPack" (
           bHigh                    := "GA1_1_OutBytes".arBytes[6],
           bLow                     := "GA1_1_OutBytes".arBytes[7],
           OUT                      := "GA1_1_Outputs".RegenValveVesselA);
NETWORK
TITLE =
      CALL  "fnWordPack" (
           bHigh                    := "GA1_1_OutBytes".arBytes[8],
           bLow                     := "GA1_1_OutBytes".arBytes[9],
           OUT                      := "GA1_1_Outputs".RegenValveVesselB);
NETWORK
TITLE =
      CALL  "fnWordPack" (
           bHigh                    := "GA1_1_OutBytes".arBytes[10],
           bLow                     := "GA1_1_OutBytes".arBytes[11],
           OUT                      := "GA1_1_Outputs".ProductionValveVesselA);
NETWORK
TITLE =
      CALL  "fnWordPack" (
           bHigh                    := "GA1_1_OutBytes".arBytes[12],
           bLow                     := "GA1_1_OutBytes".arBytes[13],
           OUT                      := "GA1_1_Outputs".ProductionValveVesselB);
NETWORK
TITLE =
      CALL  "fnWordPack" (
           bHigh                    := "GA1_1_OutBytes".arBytes[14],
           bLow                     := "GA1_1_OutBytes".arBytes[15],
           OUT                      := "GA1_1_Outputs".SolenoidValves);
NETWORK
TITLE =
      CALL  "fnWordPack" (
           bHigh                    := "GA1_1_OutBytes".arBytes[16],
           bLow                     := "GA1_1_OutBytes".arBytes[17],
           OUT                      := "GA1_1_Outputs".ConsumerValve);
NETWORK
TITLE =
      CALL  "fnWordPack" (
           bHigh                    := "GA1_1_OutBytes".arBytes[18],
           bLow                     := "GA1_1_OutBytes".arBytes[19],
           OUT                      := "GA1_1_Outputs".InletFlushingValve);
NETWORK
TITLE =
      CALL  "fnWordPack" (
           bHigh                    := "GA1_1_OutBytes".arBytes[20],
           bLow                     := "GA1_1_OutBytes".arBytes[21],
           OUT                      := "GA1_1_Outputs".ExhaustValve);
NETWORK
TITLE =
      CALL  "fnWordPack" (
           bHigh                    := "GA1_1_OutBytes".arBytes[22],
           bLow                     := "GA1_1_OutBytes".arBytes[23],
           OUT                      := "GA1_1_Outputs".Running);
NETWORK
TITLE =
      CALL  "fnWordPack" (
           bHigh                    := "GA1_1_OutBytes".arBytes[24],
           bLow                     := "GA1_1_OutBytes".arBytes[25],
           OUT                      := "GA1_1_Outputs".SecondRunning);
NETWORK
TITLE =
      CALL  "fnWordPack" (
           bHigh                    := "GA1_1_OutBytes".arBytes[26],
           bLow                     := "GA1_1_OutBytes".arBytes[27],
           OUT                      := "GA1_1_Outputs".GeneralWarning);
NETWORK
TITLE =
      CALL  "fnWordPack" (
           bHigh                    := "GA1_1_OutBytes".arBytes[28],
           bLow                     := "GA1_1_OutBytes".arBytes[29],
           OUT                      := "GA1_1_Outputs".GeneralShutdown);
END_FUNCTION_BLOCK

FUNCTION_BLOCK "GA1_2_GetOutputs"	// FB 22
VERSION : 0.1
BEGIN
NETWORK
TITLE =
      CALL  "fnWordPack" (
           bHigh                    := "GA1_2_OutBytes".arBytes[0],
           bLow                     := "GA1_2_OutBytes".arBytes[1],
           OUT                      := "GA1_2_Outputs".InletValveVesselA);
NETWORK
TITLE =
      CALL  "fnWordPack" (
           bHigh                    := "GA1_2_OutBytes".arBytes[2],
           bLow                     := "GA1_2_OutBytes".arBytes[3],
           OUT                      := "GA1_2_Outputs".InletValveVesselB);
NETWORK
TITLE =
      CALL  "fnWordPack" (
           bHigh                    := "GA1_2_OutBytes".arBytes[4],
           bLow                     := "GA1_2_OutBytes".arBytes[5],
           OUT                      := "GA1_2_Outputs".EqualizationValve);
NETWORK
TITLE =
      CALL  "fnWordPack" (
           bHigh                    := "GA1_2_OutBytes".arBytes[6],
           bLow                     := "GA1_2_OutBytes".arBytes[7],
           OUT                      := "GA1_2_Outputs".RegenValveVesselA);
NETWORK
TITLE =
      CALL  "fnWordPack" (
           bHigh                    := "GA1_2_OutBytes".arBytes[8],
           bLow                     := "GA1_2_OutBytes".arBytes[9],
           OUT                      := "GA1_2_Outputs".RegenValveVesselB);
NETWORK
TITLE =
      CALL  "fnWordPack" (
           bHigh                    := "GA1_2_OutBytes".arBytes[10],
           bLow                     := "GA1_2_OutBytes".arBytes[11],
           OUT                      := "GA1_2_Outputs".ProductionValveVesselA);
NETWORK
TITLE =
      CALL  "fnWordPack" (
           bHigh                    := "GA1_2_OutBytes".arBytes[12],
           bLow                     := "GA1_2_OutBytes".arBytes[13],
           OUT                      := "GA1_2_Outputs".ProductionValveVesselB);
NETWORK
TITLE =
      CALL  "fnWordPack" (
           bHigh                    := "GA1_2_OutBytes".arBytes[14],
           bLow                     := "GA1_2_OutBytes".arBytes[15],
           OUT                      := "GA1_2_Outputs".SolenoidValves);
NETWORK
TITLE =
      CALL  "fnWordPack" (
           bHigh                    := "GA1_2_OutBytes".arBytes[16],
           bLow                     := "GA1_2_OutBytes".arBytes[17],
           OUT                      := "GA1_2_Outputs".ConsumerValve);
NETWORK
TITLE =
      CALL  "fnWordPack" (
           bHigh                    := "GA1_2_OutBytes".arBytes[18],
           bLow                     := "GA1_2_OutBytes".arBytes[19],
           OUT                      := "GA1_2_Outputs".InletFlushingValve);
NETWORK
TITLE =
      CALL  "fnWordPack" (
           bHigh                    := "GA1_2_OutBytes".arBytes[20],
           bLow                     := "GA1_2_OutBytes".arBytes[21],
           OUT                      := "GA1_2_Outputs".ExhaustValve);
NETWORK
TITLE =
      CALL  "fnWordPack" (
           bHigh                    := "GA1_2_OutBytes".arBytes[22],
           bLow                     := "GA1_2_OutBytes".arBytes[23],
           OUT                      := "GA1_2_Outputs".Running);
NETWORK
TITLE =
      CALL  "fnWordPack" (
           bHigh                    := "GA1_2_OutBytes".arBytes[24],
           bLow                     := "GA1_2_OutBytes".arBytes[25],
           OUT                      := "GA1_2_Outputs".SecondRunning);
NETWORK
TITLE =
      CALL  "fnWordPack" (
           bHigh                    := "GA1_2_OutBytes".arBytes[26],
           bLow                     := "GA1_2_OutBytes".arBytes[27],
           OUT                      := "GA1_2_Outputs".GeneralWarning);
NETWORK
TITLE =
      CALL  "fnWordPack" (
           bHigh                    := "GA1_2_OutBytes".arBytes[28],
           bLow                     := "GA1_2_OutBytes".arBytes[29],
           OUT                      := "GA1_2_Outputs".GeneralShutdown);
END_FUNCTION_BLOCK

FUNCTION_BLOCK "GA2_1_GetOutputs"	// FB 23
VERSION : 0.1
BEGIN
NETWORK
TITLE =
      CALL  "fnWordPack" (
           bHigh                    := "GA2_1_OutBytes".arBytes[0],
           bLow                     := "GA2_1_OutBytes".arBytes[1],
           OUT                      := "GA2_1_Outputs".InletValveVesselA);
NETWORK
TITLE =
      CALL  "fnWordPack" (
           bHigh                    := "GA2_1_OutBytes".arBytes[2],
           bLow                     := "GA2_1_OutBytes".arBytes[3],
           OUT                      := "GA2_1_Outputs".InletValveVesselB);
NETWORK
TITLE =
      CALL  "fnWordPack" (
           bHigh                    := "GA2_1_OutBytes".arBytes[4],
           bLow                     := "GA2_1_OutBytes".arBytes[5],
           OUT                      := "GA2_1_Outputs".EqualizationValve);
NETWORK
TITLE =
      CALL  "fnWordPack" (
           bHigh                    := "GA2_1_OutBytes".arBytes[6],
           bLow                     := "GA2_1_OutBytes".arBytes[7],
           OUT                      := "GA2_1_Outputs".RegenValveVesselA);
NETWORK
TITLE =
      CALL  "fnWordPack" (
           bHigh                    := "GA2_1_OutBytes".arBytes[8],
           bLow                     := "GA2_1_OutBytes".arBytes[9],
           OUT                      := "GA2_1_Outputs".RegenValveVesselB);
NETWORK
TITLE =
      CALL  "fnWordPack" (
           bHigh                    := "GA2_1_OutBytes".arBytes[10],
           bLow                     := "GA2_1_OutBytes".arBytes[11],
           OUT                      := "GA2_1_Outputs".ProductionValveVesselA);
NETWORK
TITLE =
      CALL  "fnWordPack" (
           bHigh                    := "GA2_1_OutBytes".arBytes[12],
           bLow                     := "GA2_1_OutBytes".arBytes[13],
           OUT                      := "GA2_1_Outputs".ProductionValveVesselB);
NETWORK
TITLE =
      CALL  "fnWordPack" (
           bHigh                    := "GA2_1_OutBytes".arBytes[14],
           bLow                     := "GA2_1_OutBytes".arBytes[15],
           OUT                      := "GA2_1_Outputs".SolenoidValves);
NETWORK
TITLE =
      CALL  "fnWordPack" (
           bHigh                    := "GA2_1_OutBytes".arBytes[16],
           bLow                     := "GA2_1_OutBytes".arBytes[17],
           OUT                      := "GA2_1_Outputs".ConsumerValve);
NETWORK
TITLE =
      CALL  "fnWordPack" (
           bHigh                    := "GA2_1_OutBytes".arBytes[18],
           bLow                     := "GA2_1_OutBytes".arBytes[19],
           OUT                      := "GA2_1_Outputs".InletFlushingValve);
NETWORK
TITLE =
      CALL  "fnWordPack" (
           bHigh                    := "GA2_1_OutBytes".arBytes[20],
           bLow                     := "GA2_1_OutBytes".arBytes[21],
           OUT                      := "GA2_1_Outputs".ExhaustValve);
NETWORK
TITLE =
      CALL  "fnWordPack" (
           bHigh                    := "GA2_1_OutBytes".arBytes[22],
           bLow                     := "GA2_1_OutBytes".arBytes[23],
           OUT                      := "GA2_1_Outputs".Running);
NETWORK
TITLE =
      CALL  "fnWordPack" (
           bHigh                    := "GA2_1_OutBytes".arBytes[24],
           bLow                     := "GA2_1_OutBytes".arBytes[25],
           OUT                      := "GA2_1_Outputs".SecondRunning);
NETWORK
TITLE =
      CALL  "fnWordPack" (
           bHigh                    := "GA2_1_OutBytes".arBytes[26],
           bLow                     := "GA2_1_OutBytes".arBytes[27],
           OUT                      := "GA2_1_Outputs".GeneralWarning);
NETWORK
TITLE =
      CALL  "fnWordPack" (
           bHigh                    := "GA2_1_OutBytes".arBytes[28],
           bLow                     := "GA2_1_OutBytes".arBytes[29],
           OUT                      := "GA2_1_Outputs".GeneralShutdown);
END_FUNCTION_BLOCK

FUNCTION_BLOCK "GA2_2_GetOutputs"	// FB 24
VERSION : 0.1
BEGIN
NETWORK
TITLE =
      CALL  "fnWordPack" (
           bHigh                    := "GA2_2_OutBytes".arBytes[0],
           bLow                     := "GA2_2_OutBytes".arBytes[1],
           OUT                      := "GA2_2_Outputs".InletValveVesselA);
NETWORK
TITLE =
      CALL  "fnWordPack" (
           bHigh                    := "GA2_2_OutBytes".arBytes[2],
           bLow                     := "GA2_2_OutBytes".arBytes[3],
           OUT                      := "GA2_2_Outputs".InletValveVesselB);
NETWORK
TITLE =
      CALL  "fnWordPack" (
           bHigh                    := "GA2_2_OutBytes".arBytes[4],
           bLow                     := "GA2_2_OutBytes".arBytes[5],
           OUT                      := "GA2_2_Outputs".EqualizationValve);
NETWORK
TITLE =
      CALL  "fnWordPack" (
           bHigh                    := "GA2_2_OutBytes".arBytes[6],
           bLow                     := "GA2_2_OutBytes".arBytes[7],
           OUT                      := "GA2_2_Outputs".RegenValveVesselA);
NETWORK
TITLE =
      CALL  "fnWordPack" (
           bHigh                    := "GA2_2_OutBytes".arBytes[8],
           bLow                     := "GA2_2_OutBytes".arBytes[9],
           OUT                      := "GA2_2_Outputs".RegenValveVesselB);
NETWORK
TITLE =
      CALL  "fnWordPack" (
           bHigh                    := "GA2_2_OutBytes".arBytes[10],
           bLow                     := "GA2_2_OutBytes".arBytes[11],
           OUT                      := "GA2_2_Outputs".ProductionValveVesselA);
NETWORK
TITLE =
      CALL  "fnWordPack" (
           bHigh                    := "GA2_2_OutBytes".arBytes[12],
           bLow                     := "GA2_2_OutBytes".arBytes[13],
           OUT                      := "GA2_2_Outputs".ProductionValveVesselB);
NETWORK
TITLE =
      CALL  "fnWordPack" (
           bHigh                    := "GA2_2_OutBytes".arBytes[14],
           bLow                     := "GA2_2_OutBytes".arBytes[15],
           OUT                      := "GA2_2_Outputs".SolenoidValves);
NETWORK
TITLE =
      CALL  "fnWordPack" (
           bHigh                    := "GA2_2_OutBytes".arBytes[16],
           bLow                     := "GA2_2_OutBytes".arBytes[17],
           OUT                      := "GA2_2_Outputs".ConsumerValve);
NETWORK
TITLE =
      CALL  "fnWordPack" (
           bHigh                    := "GA2_2_OutBytes".arBytes[18],
           bLow                     := "GA2_2_OutBytes".arBytes[19],
           OUT                      := "GA2_2_Outputs".InletFlushingValve);
NETWORK
TITLE =
      CALL  "fnWordPack" (
           bHigh                    := "GA2_2_OutBytes".arBytes[20],
           bLow                     := "GA2_2_OutBytes".arBytes[21],
           OUT                      := "GA2_2_Outputs".ExhaustValve);
NETWORK
TITLE =
      CALL  "fnWordPack" (
           bHigh                    := "GA2_2_OutBytes".arBytes[22],
           bLow                     := "GA2_2_OutBytes".arBytes[23],
           OUT                      := "GA2_2_Outputs".Running);
NETWORK
TITLE =
      CALL  "fnWordPack" (
           bHigh                    := "GA2_2_OutBytes".arBytes[24],
           bLow                     := "GA2_2_OutBytes".arBytes[25],
           OUT                      := "GA2_2_Outputs".SecondRunning);
NETWORK
TITLE =
      CALL  "fnWordPack" (
           bHigh                    := "GA2_2_OutBytes".arBytes[26],
           bLow                     := "GA2_2_OutBytes".arBytes[27],
           OUT                      := "GA2_2_Outputs".GeneralWarning);
NETWORK
TITLE =
      CALL  "fnWordPack" (
           bHigh                    := "GA2_2_OutBytes".arBytes[28],
           bLow                     := "GA2_2_OutBytes".arBytes[29],
           OUT                      := "GA2_2_Outputs".GeneralShutdown);
END_FUNCTION_BLOCK

FUNCTION_BLOCK "ModbusStartStop"	// FB 25
VERSION : 0.1
VAR_TEMP
  xAlwaysOn : BOOL ;
END_VAR
BEGIN
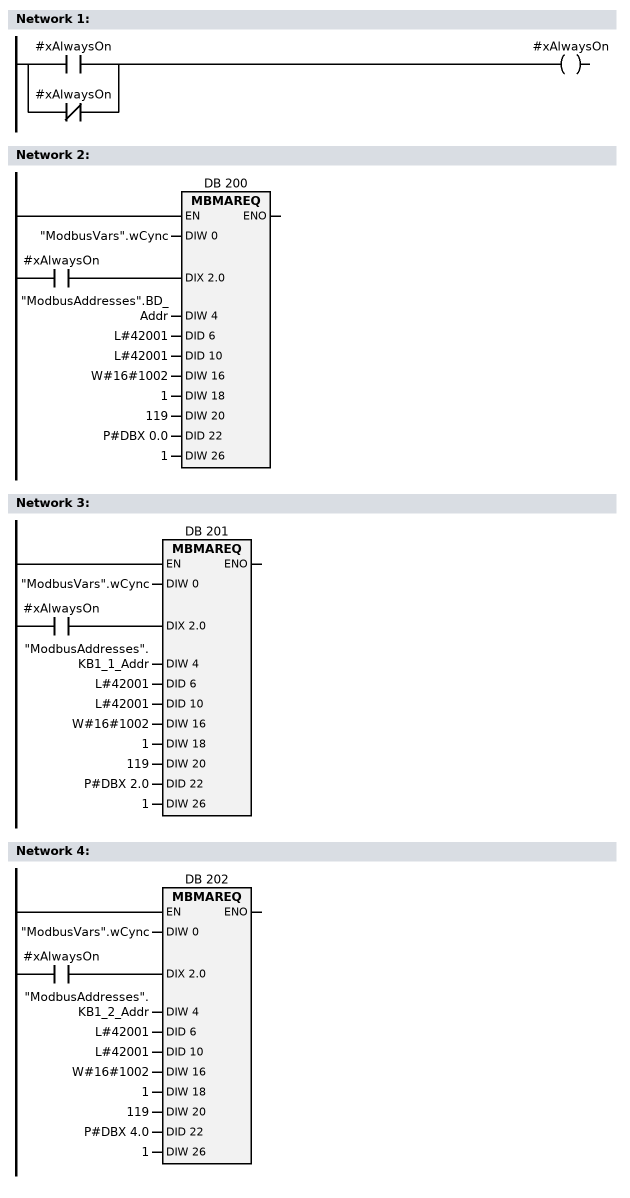
NETWORK
TITLE =
      O     #xAlwaysOn;
      ON    #xAlwaysOn;
      =     #xAlwaysOn;
NETWORK
TITLE =
      A     #xAlwaysOn;
      =     L 1.0;
      BLD   103;
      CALL  "MBMAREQ" , DB 200 (
           DIW 0                    := "ModbusVars".wCync,
           DIX 2.0                  := L 1.0,
           DIW 4                    := "ModbusAddresses".BD_Addr,
           DID 6                    := L#42001,
           DID 10                   := L#42001,
           DIW 16                   := W#16#1002,
           DIW 18                   := 1,
           DIW 20                   := 119,
           DID 22                   := P#DBX 0.0,
           DIW 26                   := 1);
      NOP   0;
NETWORK
TITLE =
      A     #xAlwaysOn;
      =     L 1.0;
      BLD   103;
      CALL  "MBMAREQ" , DB 201 (
           DIW 0                    := "ModbusVars".wCync,
           DIX 2.0                  := L 1.0,
           DIW 4                    := "ModbusAddresses".KB1_1_Addr,
           DID 6                    := L#42001,
           DID 10                   := L#42001,
           DIW 16                   := W#16#1002,
           DIW 18                   := 1,
           DIW 20                   := 119,
           DID 22                   := P#DBX 2.0,
           DIW 26                   := 1);
      NOP   0;
NETWORK
TITLE =
      A     #xAlwaysOn;
      =     L 1.0;
      BLD   103;
      CALL  "MBMAREQ" , DB 202 (
           DIW 0                    := "ModbusVars".wCync,
           DIX 2.0                  := L 1.0,
           DIW 4                    := "ModbusAddresses".KB1_2_Addr,
           DID 6                    := L#42001,
           DID 10                   := L#42001,
           DIW 16                   := W#16#1002,
           DIW 18                   := 1,
           DIW 20                   := 119,
           DID 22                   := P#DBX 4.0,
           DIW 26                   := 1);
      NOP   0;
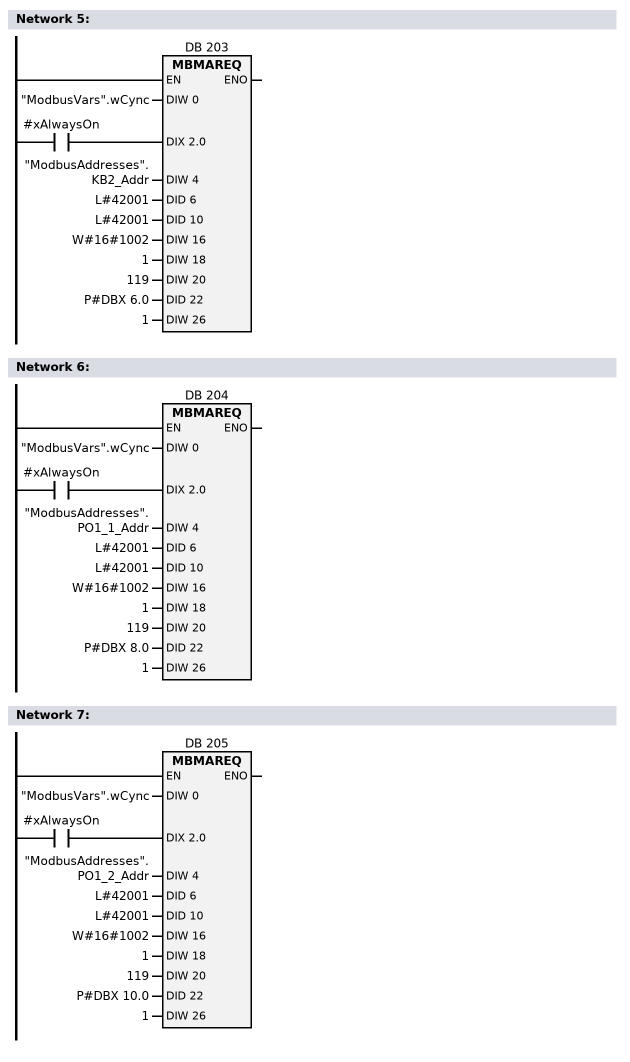
NETWORK
TITLE =
      A     #xAlwaysOn;
      =     L 1.0;
      BLD   103;
      CALL  "MBMAREQ" , DB 203 (
           DIW 0                    := "ModbusVars".wCync,
           DIX 2.0                  := L 1.0,
           DIW 4                    := "ModbusAddresses".KB2_Addr,
           DID 6                    := L#42001,
           DID 10                   := L#42001,
           DIW 16                   := W#16#1002,
           DIW 18                   := 1,
           DIW 20                   := 119,
           DID 22                   := P#DBX 6.0,
           DIW 26                   := 1);
      NOP   0;
NETWORK
TITLE =
      A     #xAlwaysOn;
      =     L 1.0;
      BLD   103;
      CALL  "MBMAREQ" , DB 204 (
           DIW 0                    := "ModbusVars".wCync,
           DIX 2.0                  := L 1.0,
           DIW 4                    := "ModbusAddresses".PO1_1_Addr,
           DID 6                    := L#42001,
           DID 10                   := L#42001,
           DIW 16                   := W#16#1002,
           DIW 18                   := 1,
           DIW 20                   := 119,
           DID 22                   := P#DBX 8.0,
           DIW 26                   := 1);
      NOP   0;
NETWORK
TITLE =
      A     #xAlwaysOn;
      =     L 1.0;
      BLD   103;
      CALL  "MBMAREQ" , DB 205 (
           DIW 0                    := "ModbusVars".wCync,
           DIX 2.0                  := L 1.0,
           DIW 4                    := "ModbusAddresses".PO1_2_Addr,
           DID 6                    := L#42001,
           DID 10                   := L#42001,
           DIW 16                   := W#16#1002,
           DIW 18                   := 1,
           DIW 20                   := 119,
           DID 22                   := P#DBX 10.0,
           DIW 26                   := 1);
      NOP   0;
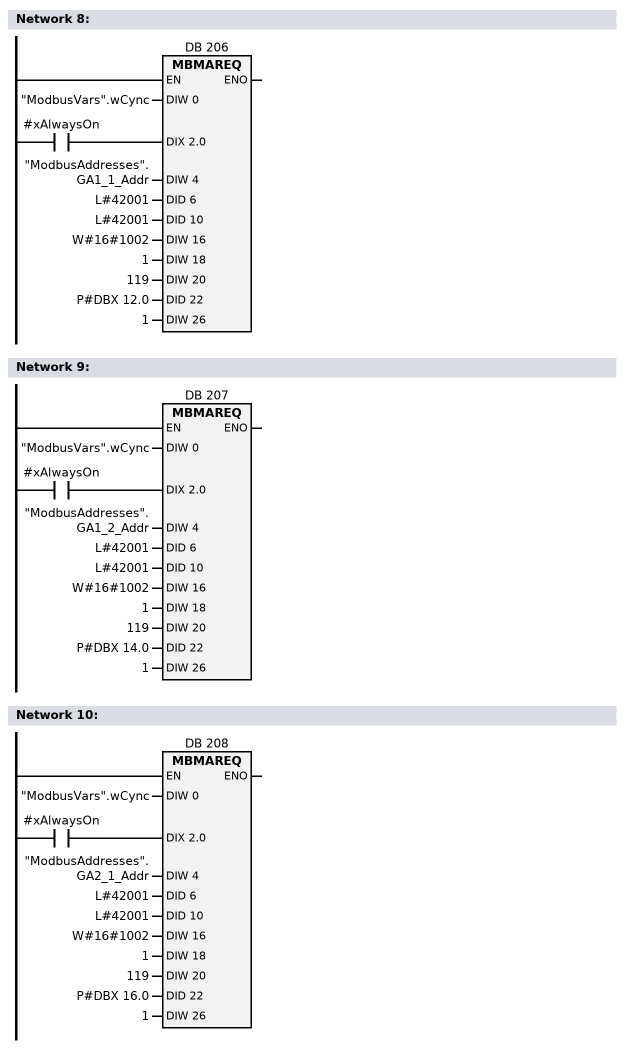
NETWORK
TITLE =
      A     #xAlwaysOn;
      =     L 1.0;
      BLD   103;
      CALL  "MBMAREQ" , DB 206 (
           DIW 0                    := "ModbusVars".wCync,
           DIX 2.0                  := L 1.0,
           DIW 4                    := "ModbusAddresses".GA1_1_Addr,
           DID 6                    := L#42001,
           DID 10                   := L#42001,
           DIW 16                   := W#16#1002,
           DIW 18                   := 1,
           DIW 20                   := 119,
           DID 22                   := P#DBX 12.0,
           DIW 26                   := 1);
      NOP   0;
NETWORK
TITLE =
      A     #xAlwaysOn;
      =     L 1.0;
      BLD   103;
      CALL  "MBMAREQ" , DB 207 (
           DIW 0                    := "ModbusVars".wCync,
           DIX 2.0                  := L 1.0,
           DIW 4                    := "ModbusAddresses".GA1_2_Addr,
           DID 6                    := L#42001,
           DID 10                   := L#42001,
           DIW 16                   := W#16#1002,
           DIW 18                   := 1,
           DIW 20                   := 119,
           DID 22                   := P#DBX 14.0,
           DIW 26                   := 1);
      NOP   0;
NETWORK
TITLE =
      A     #xAlwaysOn;
      =     L 1.0;
      BLD   103;
      CALL  "MBMAREQ" , DB 208 (
           DIW 0                    := "ModbusVars".wCync,
           DIX 2.0                  := L 1.0,
           DIW 4                    := "ModbusAddresses".GA2_1_Addr,
           DID 6                    := L#42001,
           DID 10                   := L#42001,
           DIW 16                   := W#16#1002,
           DIW 18                   := 1,
           DIW 20                   := 119,
           DID 22                   := P#DBX 16.0,
           DIW 26                   := 1);
      NOP   0;
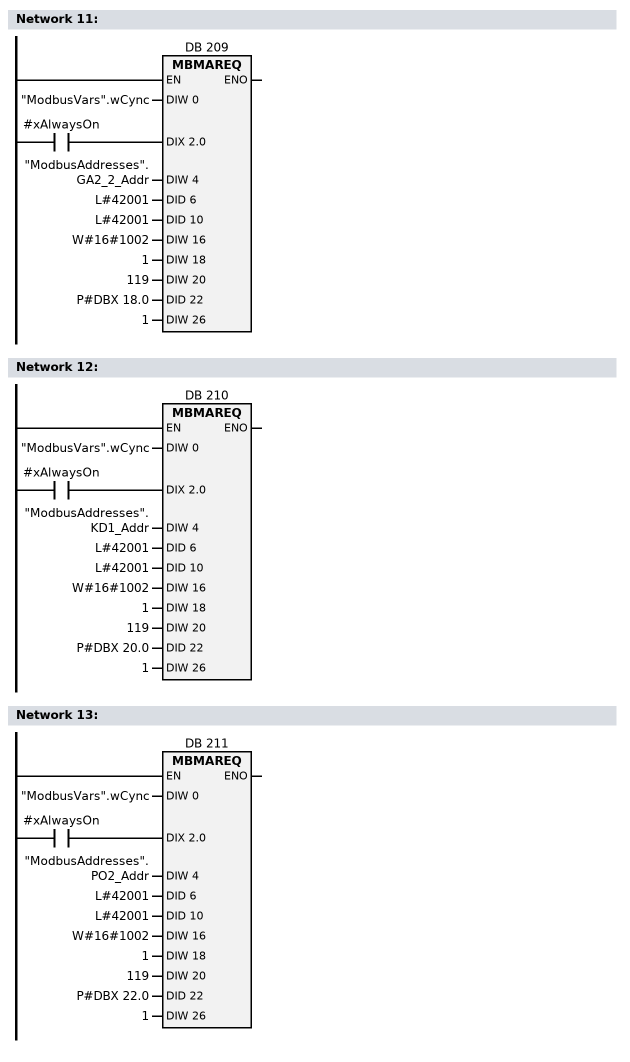
NETWORK
TITLE =
      A     #xAlwaysOn;
      =     L 1.0;
      BLD   103;
      CALL  "MBMAREQ" , DB 209 (
           DIW 0                    := "ModbusVars".wCync,
           DIX 2.0                  := L 1.0,
           DIW 4                    := "ModbusAddresses".GA2_2_Addr,
           DID 6                    := L#42001,
           DID 10                   := L#42001,
           DIW 16                   := W#16#1002,
           DIW 18                   := 1,
           DIW 20                   := 119,
           DID 22                   := P#DBX 18.0,
           DIW 26                   := 1);
      NOP   0;
NETWORK
TITLE =
      A     #xAlwaysOn;
      =     L 1.0;
      BLD   103;
      CALL  "MBMAREQ" , DB 210 (
           DIW 0                    := "ModbusVars".wCync,
           DIX 2.0                  := L 1.0,
           DIW 4                    := "ModbusAddresses".KD1_Addr,
           DID 6                    := L#42001,
           DID 10                   := L#42001,
           DIW 16                   := W#16#1002,
           DIW 18                   := 1,
           DIW 20                   := 119,
           DID 22                   := P#DBX 20.0,
           DIW 26                   := 1);
      NOP   0;
NETWORK
TITLE =
      A     #xAlwaysOn;
      =     L 1.0;
      BLD   103;
      CALL  "MBMAREQ" , DB 211 (
           DIW 0                    := "ModbusVars".wCync,
           DIX 2.0                  := L 1.0,
           DIW 4                    := "ModbusAddresses".PO2_Addr,
           DID 6                    := L#42001,
           DID 10                   := L#42001,
           DIW 16                   := W#16#1002,
           DIW 18                   := 1,
           DIW 20                   := 119,
           DID 22                   := P#DBX 22.0,
           DIW 26                   := 1);
      NOP   0;
END_FUNCTION_BLOCK

FUNCTION_BLOCK "GetStartStopBytes"	// FB 26
VERSION : 0.1
BEGIN
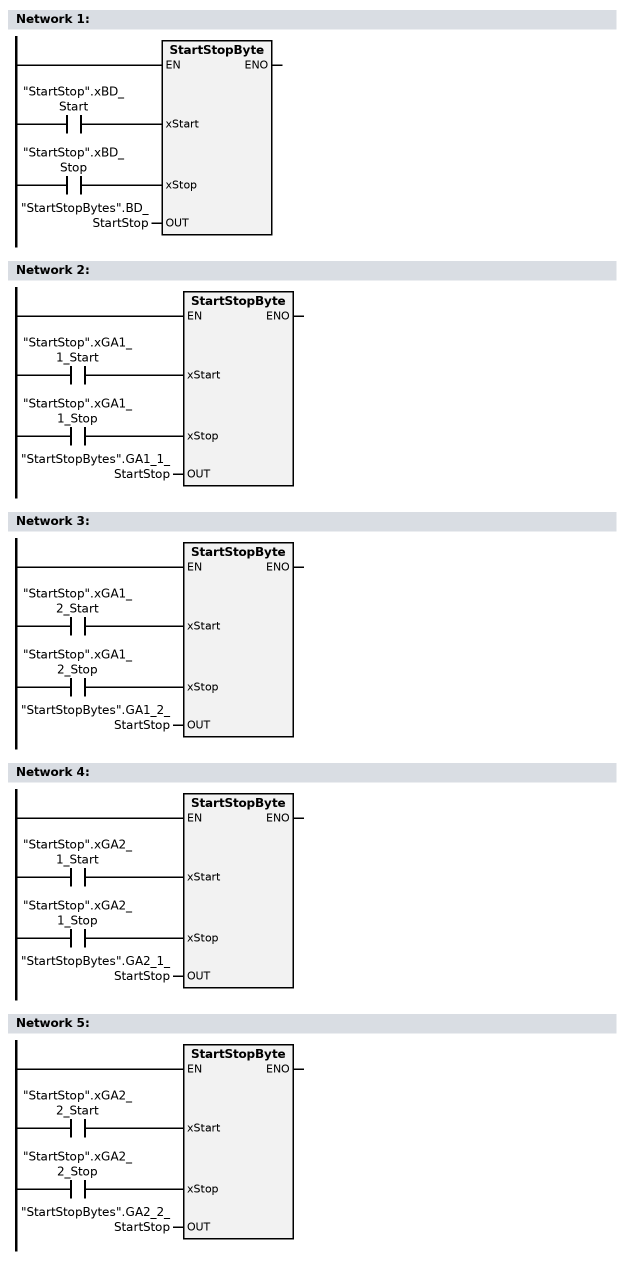
NETWORK
TITLE =
      A     "StartStop".xBD_Start;
      =     L 0.0;
      BLD   103;
      A     "StartStop".xBD_Stop;
      =     L 0.1;
      BLD   103;
      CALL  "StartStopByte" (
           xStart                   := L 0.0,
           xStop                    := L 0.1,
           OUT                      := "StartStopBytes".BD_StartStop);
      NOP   0;
NETWORK
TITLE =
      A     "StartStop".xGA1_1_Start;
      =     L 0.0;
      BLD   103;
      A     "StartStop".xGA1_1_Stop;
      =     L 0.1;
      BLD   103;
      CALL  "StartStopByte" (
           xStart                   := L 0.0,
           xStop                    := L 0.1,
           OUT                      := "StartStopBytes".GA1_1_StartStop);
      NOP   0;
NETWORK
TITLE =
      A     "StartStop".xGA1_2_Start;
      =     L 0.0;
      BLD   103;
      A     "StartStop".xGA1_2_Stop;
      =     L 0.1;
      BLD   103;
      CALL  "StartStopByte" (
           xStart                   := L 0.0,
           xStop                    := L 0.1,
           OUT                      := "StartStopBytes".GA1_2_StartStop);
      NOP   0;
NETWORK
TITLE =
      A     "StartStop".xGA2_1_Start;
      =     L 0.0;
      BLD   103;
      A     "StartStop".xGA2_1_Stop;
      =     L 0.1;
      BLD   103;
      CALL  "StartStopByte" (
           xStart                   := L 0.0,
           xStop                    := L 0.1,
           OUT                      := "StartStopBytes".GA2_1_StartStop);
      NOP   0;
NETWORK
TITLE =
      A     "StartStop".xGA2_2_Start;
      =     L 0.0;
      BLD   103;
      A     "StartStop".xGA2_2_Stop;
      =     L 0.1;
      BLD   103;
      CALL  "StartStopByte" (
           xStart                   := L 0.0,
           xStop                    := L 0.1,
           OUT                      := "StartStopBytes".GA2_2_StartStop);
      NOP   0;
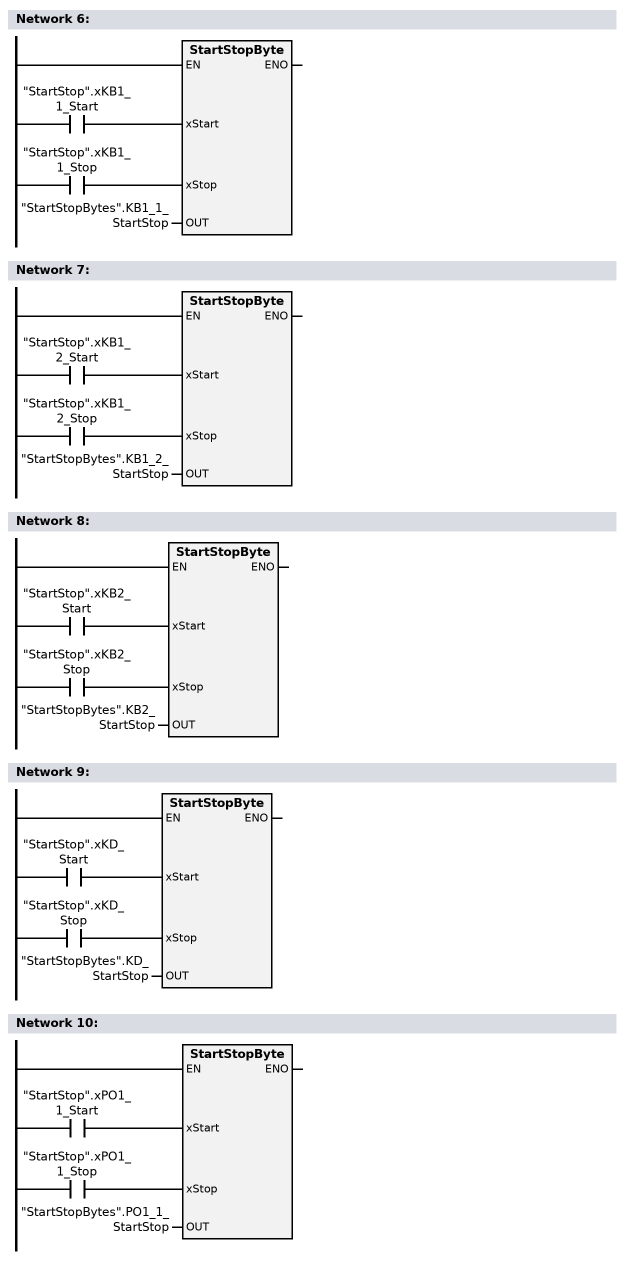
NETWORK
TITLE =
      A     "StartStop".xKB1_1_Start;
      =     L 0.0;
      BLD   103;
      A     "StartStop".xKB1_1_Stop;
      =     L 0.1;
      BLD   103;
      CALL  "StartStopByte" (
           xStart                   := L 0.0,
           xStop                    := L 0.1,
           OUT                      := "StartStopBytes".KB1_1_StartStop);
      NOP   0;
NETWORK
TITLE =
      A     "StartStop".xKB1_2_Start;
      =     L 0.0;
      BLD   103;
      A     "StartStop".xKB1_2_Stop;
      =     L 0.1;
      BLD   103;
      CALL  "StartStopByte" (
           xStart                   := L 0.0,
           xStop                    := L 0.1,
           OUT                      := "StartStopBytes".KB1_2_StartStop);
      NOP   0;
NETWORK
TITLE =
      A     "StartStop".xKB2_Start;
      =     L 0.0;
      BLD   103;
      A     "StartStop".xKB2_Stop;
      =     L 0.1;
      BLD   103;
      CALL  "StartStopByte" (
           xStart                   := L 0.0,
           xStop                    := L 0.1,
           OUT                      := "StartStopBytes".KB2_StartStop);
      NOP   0;
NETWORK
TITLE =
      A     "StartStop".xKD_Start;
      =     L 0.0;
      BLD   103;
      A     "StartStop".xKD_Stop;
      =     L 0.1;
      BLD   103;
      CALL  "StartStopByte" (
           xStart                   := L 0.0,
           xStop                    := L 0.1,
           OUT                      := "StartStopBytes".KD_StartStop);
      NOP   0;
NETWORK
TITLE =
      A     "StartStop".xPO1_1_Start;
      =     L 0.0;
      BLD   103;
      A     "StartStop".xPO1_1_Stop;
      =     L 0.1;
      BLD   103;
      CALL  "StartStopByte" (
           xStart                   := L 0.0,
           xStop                    := L 0.1,
           OUT                      := "StartStopBytes".PO1_1_StartStop);
      NOP   0;
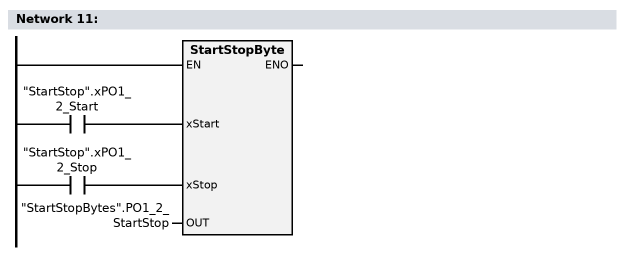
NETWORK
TITLE =
      A     "StartStop".xPO1_2_Start;
      =     L 0.0;
      BLD   103;
      A     "StartStop".xPO1_2_Stop;
      =     L 0.1;
      BLD   103;
      CALL  "StartStopByte" (
           xStart                   := L 0.0,
           xStop                    := L 0.1,
           OUT                      := "StartStopBytes".PO1_2_StartStop);
      NOP   0;
END_FUNCTION_BLOCK

FUNCTION_BLOCK "GetAll"	// FB 27
VERSION : 0.1
BEGIN
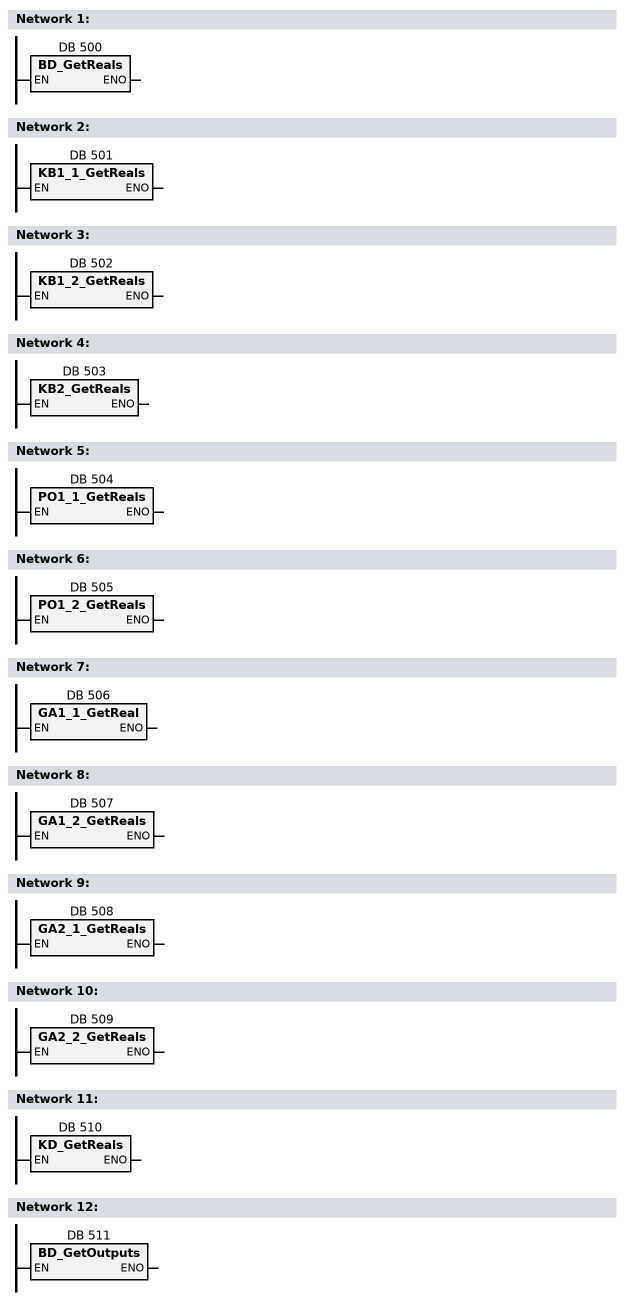
NETWORK
TITLE =
      CALL  "BD_GetReals" , DB 500;
      NOP   0;
NETWORK
TITLE =
      CALL  "KB1_1_GetReals" , DB 501;
      NOP   0;
NETWORK
TITLE =
      CALL  "KB1_2_GetReals" , DB 502;
      NOP   0;
NETWORK
TITLE =
      CALL  "KB2_GetReals" , DB 503;
      NOP   0;
NETWORK
TITLE =
      CALL  "PO1_1_GetReals" , DB 504;
      NOP   0;
NETWORK
TITLE =
      CALL  "PO1_2_GetReals" , DB 505;
      NOP   0;
NETWORK
TITLE =
      CALL  "GA1_1_GetReal" , DB 506;
      NOP   0;
NETWORK
TITLE =
      CALL  "GA1_2_GetReals" , DB 507;
      NOP   0;
NETWORK
TITLE =
      CALL  "GA2_1_GetReals" , DB 508;
      NOP   0;
NETWORK
TITLE =
      CALL  "GA2_2_GetReals" , DB 509;
      NOP   0;
NETWORK
TITLE =
      CALL  "KD_GetReals" , DB 510;
      NOP   0;
NETWORK
TITLE =
      CALL  "BD_GetOutputs" , DB 511;
      NOP   0;
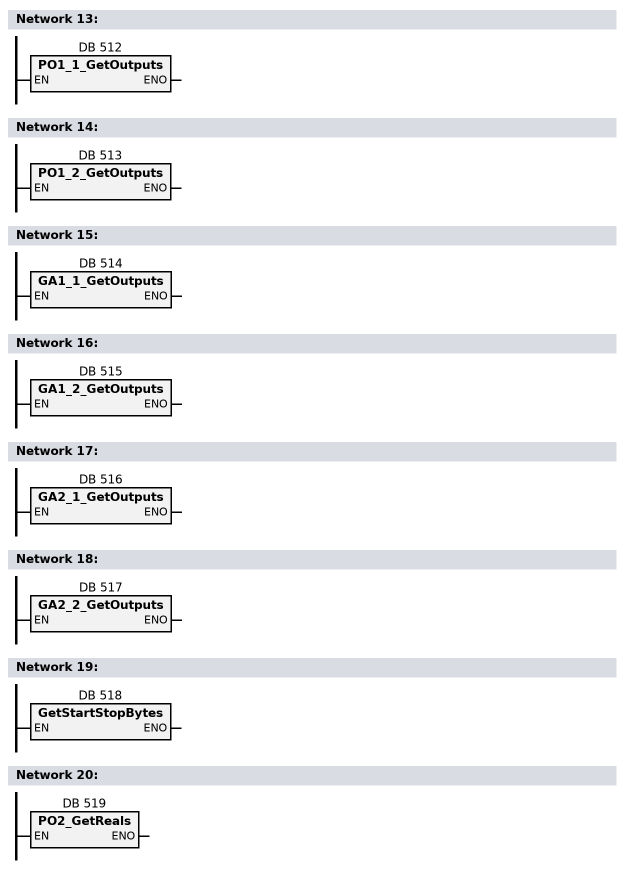
NETWORK
TITLE =
      CALL  "PO1_1_GetOutputs" , DB 512;
      NOP   0;
NETWORK
TITLE =
      CALL  "PO1_2_GetOutputs" , DB 513;
      NOP   0;
NETWORK
TITLE =
      CALL  "GA1_1_GetOutputs" , DB 514;
      NOP   0;
NETWORK
TITLE =
      CALL  "GA1_2_GetOutputs" , DB 515;
      NOP   0;
NETWORK
TITLE =
      CALL  "GA2_1_GetOutputs" , DB 516;
      NOP   0;
NETWORK
TITLE =
      CALL  "GA2_2_GetOutputs" , DB 517;
      NOP   0;
NETWORK
TITLE =
      CALL  "GetStartStopBytes" , DB 518;
      NOP   0;
NETWORK
TITLE =
      CALL  "PO2_GetReals" , DB 519;
      NOP   0;
END_FUNCTION_BLOCK

FUNCTION_BLOCK "ModbusAll"	// FB 28
VERSION : 0.1
BEGIN
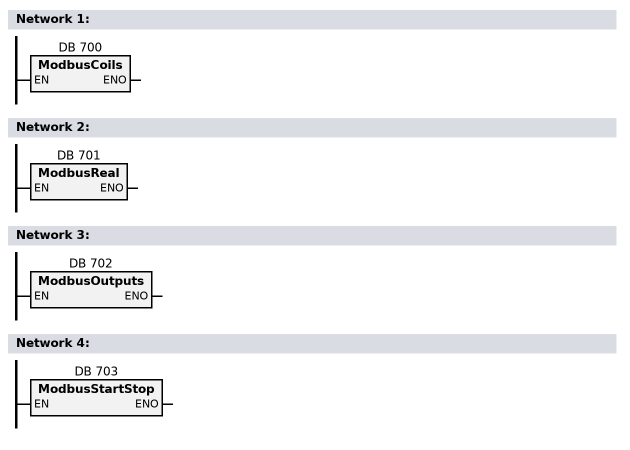
NETWORK
TITLE =
      CALL  "ModbusCoils" , DB 700;
      NOP   0;
NETWORK
TITLE =
      CALL  "ModbusReal" , DB 701;
      NOP   0;
NETWORK
TITLE =
      CALL  "ModbusOutputs" , DB 702;
      NOP   0;
NETWORK
TITLE =
      CALL  "ModbusStartStop" , DB 703;
      NOP   0;
END_FUNCTION_BLOCK

FUNCTION_BLOCK "InToVars"	// FB 29
VERSION : 0.1
VAR_TEMP
  xError : BOOL ;
END_VAR
BEGIN
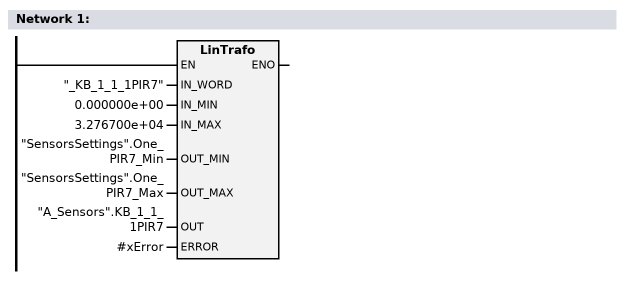
NETWORK
TITLE =
      CALL  "LinTrafo" (
           IN_WORD                  := "_KB_1_1_1PIR7",
           IN_MIN                   := 0.000000e+00,
           IN_MAX                   := 3.276700e+04,
           OUT_MIN                  := "SensorsSettings".One_PIR7_Min,
           OUT_MAX                  := "SensorsSettings".One_PIR7_Max,
           OUT                      := "A_Sensors".KB_1_1_1PIR7,
           ERROR                    := #xError);
      NOP   0;
END_FUNCTION_BLOCK

FUNCTION_BLOCK "InToVarsST"	// FB 30
VERSION : 0.1
VAR_TEMP
  xError : BOOL ;
END_VAR
BEGIN
NETWORK
TITLE =
      CALL  "LinTrafo" (
           IN_WORD                  := PIW 256,
           IN_MIN                   := 0.000000e+00,
           IN_MAX                   := 2.764000e+04,
           OUT_MIN                  := "SensorsSettings".One_PIR7_Min,
           OUT_MAX                  := "SensorsSettings".One_PIR7_Max,
           OUT                      := "A_Sensors".KB_1_1_1PIR7,
           ERROR                    := #xError);
NETWORK
TITLE =
      CALL  "LinTrafo" (
           IN_WORD                  := PIW 258,
           IN_MIN                   := 0.000000e+00,
           IN_MAX                   := 2.764000e+04,
           OUT_MIN                  := "SensorsSettings".Two_PIR7_Min,
           OUT_MAX                  := "SensorsSettings".Two_PIR7_Max,
           OUT                      := "A_Sensors".KB_1_2_2PIR7,
           ERROR                    := #xError);
NETWORK
TITLE =
      CALL  "LinTrafo" (
           IN_WORD                  := PIW 260,
           IN_MIN                   := 0.000000e+00,
           IN_MAX                   := 2.764000e+04,
           OUT_MIN                  := "SensorsSettings".One_PIR6_Min,
           OUT_MAX                  := "SensorsSettings".One_PIR6_Max,
           OUT                      := "A_Sensors".KZA_1_1_1PIR6,
           ERROR                    := #xError);
NETWORK
TITLE =
      CALL  "LinTrafo" (
           IN_WORD                  := PIW 262,
           IN_MIN                   := 0.000000e+00,
           IN_MAX                   := 2.764000e+04,
           OUT_MIN                  := "SensorsSettings".Two_PIR6_Min,
           OUT_MAX                  := "SensorsSettings".Two_PIR6_Max,
           OUT                      := "A_Sensors".KZA_1_2_2PIR6,
           ERROR                    := #xError);
NETWORK
TITLE =
      CALL  "LinTrafo" (
           IN_WORD                  := PIW 264,
           IN_MIN                   := 0.000000e+00,
           IN_MAX                   := 2.764000e+04,
           OUT_MIN                  := "SensorsSettings".PIR8_Min,
           OUT_MAX                  := "SensorsSettings".PIR8_Max,
           OUT                      := "A_Sensors".KB_2_PIR8,
           ERROR                    := #xError);
NETWORK
TITLE =
      CALL  "LinTrafo" (
           IN_WORD                  := PIW 266,
           IN_MIN                   := 0.000000e+00,
           IN_MAX                   := 2.764000e+04,
           OUT_MIN                  := "SensorsSettings".One_PIR20_Min,
           OUT_MAX                  := "SensorsSettings".One_PIR20_Max,
           OUT                      := "A_Sensors".One_PIR20,
           ERROR                    := #xError);
NETWORK
TITLE =
      CALL  "LinTrafo" (
           IN_WORD                  := PIW 268,
           IN_MIN                   := 0.000000e+00,
           IN_MAX                   := 2.764000e+04,
           OUT_MIN                  := "SensorsSettings".Two_PIR20_Min,
           OUT_MAX                  := "SensorsSettings".Two_PIR20_Max,
           OUT                      := "A_Sensors".KZA_2_2_2PIR20,
           ERROR                    := #xError);
NETWORK
TITLE =
      CALL  "LinTrafo" (
           IN_WORD                  := PIW 304,
           IN_MIN                   := 0.000000e+00,
           IN_MAX                   := 2.764000e+04,
           OUT_MIN                  := "SensorsSettings".TIR10_Min,
           OUT_MAX                  := "SensorsSettings".TIR10_Max,
           OUT                      := "A_Sensors".TIR10,
           ERROR                    := #xError);
NETWORK
TITLE =
      CALL  "LinTrafo" (
           IN_WORD                  := PIW 272,
           IN_MIN                   := 0.000000e+00,
           IN_MAX                   := 2.764000e+04,
           OUT_MIN                  := "SensorsSettings".FIR10_Min,
           OUT_MAX                  := "SensorsSettings".FIR10_Max,
           OUT                      := "A_Sensors".FIR10,
           ERROR                    := #xError);
NETWORK
TITLE =
      CALL  "LinTrafo" (
           IN_WORD                  := PIW 274,
           IN_MIN                   := 0.000000e+00,
           IN_MAX                   := 2.764000e+04,
           OUT_MIN                  := "SensorsSettings".PIR5_Min,
           OUT_MAX                  := "SensorsSettings".PIR5_Max,
           OUT                      := "A_Sensors".PIR5,
           ERROR                    := #xError);
NETWORK
TITLE =
      CALL  "LinTrafo" (
           IN_WORD                  := PIW 276,
           IN_MIN                   := 0.000000e+00,
           IN_MAX                   := 2.764000e+04,
           OUT_MIN                  := "SensorsSettings".FIR5_Min,
           OUT_MAX                  := "SensorsSettings".FIR5_Max,
           OUT                      := "A_Sensors".FIR5,
           ERROR                    := #xError);
NETWORK
TITLE =
      CALL  "LinTrafo" (
           IN_WORD                  := PIW 278,
           IN_MIN                   := 0.000000e+00,
           IN_MAX                   := 2.764000e+04,
           OUT_MIN                  := "SensorsSettings".PIRC21_Min,
           OUT_MAX                  := "SensorsSettings".PIRC21_Max,
           OUT                      := "A_Sensors".PIRC21,
           ERROR                    := #xError);
NETWORK
TITLE =
      CALL  "LinTrafo" (
           IN_WORD                  := PIW 280,
           IN_MIN                   := 0.000000e+00,
           IN_MAX                   := 2.764000e+04,
           OUT_MIN                  := "SensorsSettings".One_PIR27_Min,
           OUT_MAX                  := "SensorsSettings".One_PIR27_Max,
           OUT                      := "A_Sensors".One_PIR27,
           ERROR                    := #xError);
NETWORK
TITLE =
      CALL  "LinTrafo" (
           IN_WORD                  := PIW 282,
           IN_MIN                   := 0.000000e+00,
           IN_MAX                   := 2.764000e+04,
           OUT_MIN                  := "SensorsSettings".QIRAH3_Min,
           OUT_MAX                  := "SensorsSettings".QIRAH3_Max,
           OUT                      := "A_Sensors".QIRAH3,
           ERROR                    := #xError);
NETWORK
TITLE =
      CALL  "LinTrafo" (
           IN_WORD                  := PIW 284,
           IN_MIN                   := 0.000000e+00,
           IN_MAX                   := 2.764000e+04,
           OUT_MIN                  := "SensorsSettings".Two_PIR27_Min,
           OUT_MAX                  := "SensorsSettings".Two_PIR27_Max,
           OUT                      := "A_Sensors".Two_PIR27,
           ERROR                    := #xError);
NETWORK
TITLE =
      CALL  "LinTrafo" (
           IN_WORD                  := PIW 286,
           IN_MIN                   := 0.000000e+00,
           IN_MAX                   := 2.764000e+04,
           OUT_MIN                  := "SensorsSettings".PIR4_Min,
           OUT_MAX                  := "SensorsSettings".PIR4_Max,
           OUT                      := "A_Sensors".PIR4,
           ERROR                    := #xError);
NETWORK
TITLE =
      CALL  "LinTrafo" (
           IN_WORD                  := PIW 288,
           IN_MIN                   := 0.000000e+00,
           IN_MAX                   := 2.764000e+04,
           OUT_MIN                  := "SensorsSettings".FIR_4_Min,
           OUT_MAX                  := "SensorsSettings".FIR_4_Max,
           OUT                      := "A_Sensors".FIR_4,
           ERROR                    := #xError);
NETWORK
TITLE =
      CALL  "LinTrafo" (
           IN_WORD                  := PIW 290,
           IN_MIN                   := 0.000000e+00,
           IN_MAX                   := 2.764000e+04,
           OUT_MIN                  := "SensorsSettings".PIRC22_Min,
           OUT_MAX                  := "SensorsSettings".PIRC22_Max,
           OUT                      := "A_Sensors".PIRC22,
           ERROR                    := #xError);
NETWORK
TITLE =
      CALL  "LinTrafo" (
           IN_WORD                  := PIW 292,
           IN_MIN                   := 0.000000e+00,
           IN_MAX                   := 2.764000e+04,
           OUT_MIN                  := "SensorsSettings".PIRC23_Min,
           OUT_MAX                  := "SensorsSettings".PIRC23_Max,
           OUT                      := "A_Sensors".PIRC23,
           ERROR                    := #xError);
NETWORK
TITLE =
      CALL  "LinTrafo" (
           IN_WORD                  := PIW 294,
           IN_MIN                   := 0.000000e+00,
           IN_MAX                   := 2.764000e+04,
           OUT_MIN                  := "SensorsSettings".PIRC24_Min,
           OUT_MAX                  := "SensorsSettings".PIRC24_Max,
           OUT                      := "A_Sensors".PIRC24,
           ERROR                    := #xError);
NETWORK
TITLE =
      CALL  "LinTrafo" (
           IN_WORD                  := PIW 296,
           IN_MIN                   := 0.000000e+00,
           IN_MAX                   := 2.764000e+04,
           OUT_MIN                  := "SensorsSettings".PIRC25_Min,
           OUT_MAX                  := "SensorsSettings".PIRC25_Max,
           OUT                      := "A_Sensors".PIRC25,
           ERROR                    := #xError);
NETWORK
TITLE =
      CALL  "LinTrafo" (
           IN_WORD                  := PIW 298,
           IN_MIN                   := 0.000000e+00,
           IN_MAX                   := 2.764000e+04,
           OUT_MIN                  := "SensorsSettings".FIR_25_Min,
           OUT_MAX                  := "SensorsSettings".FIR_25_Max,
           OUT                      := "A_Sensors".FIR_25,
           ERROR                    := #xError);
NETWORK
TITLE =
      CALL  "LinTrafo" (
           IN_WORD                  := PIW 300,
           IN_MIN                   := 0.000000e+00,
           IN_MAX                   := 2.764000e+04,
           OUT_MIN                  := "SensorsSettings".One_PIRC26_Min,
           OUT_MAX                  := "SensorsSettings".One_PIRC26_Max,
           OUT                      := "A_Sensors".One_PIRC26,
           ERROR                    := #xError);
NETWORK
TITLE =
      CALL  "LinTrafo" (
           IN_WORD                  := PIW 302,
           IN_MIN                   := 0.000000e+00,
           IN_MAX                   := 2.764000e+04,
           OUT_MIN                  := "SensorsSettings".Two_PIRC26_Min,
           OUT_MAX                  := "SensorsSettings".Two_PIRC26_Max,
           OUT                      := "A_Sensors".Two_PIRC26,
           ERROR                    := #xError);
NETWORK
TITLE =
      CALL  "LinTrafo" (
           IN_WORD                  := PIW 270,
           IN_MIN                   := 0.000000e+00,
           IN_MAX                   := 2.764000e+04,
           OUT_MIN                  := "SensorsSettings".PIRC_C10_Min,
           OUT_MAX                  := "SensorsSettings".PIRC_C10_Max,
           OUT                      := "A_Sensors".PIRC_C10,
           ERROR                    := #xError);
NETWORK
TITLE =
      CALL  "LinTrafo" (
           IN_WORD                  := PIW 306,
           IN_MIN                   := 0.000000e+00,
           IN_MAX                   := 2.764000e+04,
           OUT_MIN                  := "SensorsSettings".TIR5_Min,
           OUT_MAX                  := "SensorsSettings".TIR5_Max,
           OUT                      := "A_Sensors".TIR5,
           ERROR                    := #xError);
NETWORK
TITLE =
      CALL  "LinTrafo" (
           IN_WORD                  := PIW 308,
           IN_MIN                   := 0.000000e+00,
           IN_MAX                   := 2.764000e+04,
           OUT_MIN                  := "SensorsSettings".TIR4_Min,
           OUT_MAX                  := "SensorsSettings".TIR4_Max,
           OUT                      := "A_Sensors".TIR4,
           ERROR                    := #xError);
NETWORK
TITLE =
      CALL  "LinTrafo" (
           IN_WORD                  := PIW 310,
           IN_MIN                   := 0.000000e+00,
           IN_MAX                   := 2.764000e+04,
           OUT_MIN                  := "SensorsSettings".TIR25_Min,
           OUT_MAX                  := "SensorsSettings".TIR25_Max,
           OUT                      := "A_Sensors".TIR25,
           ERROR                    := #xError);
NETWORK
TITLE =
      CALL  "LinTrafo" (
           IN_WORD                  := PIW 312,
           IN_MIN                   := 0.000000e+00,
           IN_MAX                   := 2.764000e+04,
           OUT_MIN                  := "SensorsSettings".AIR1_Min,
           OUT_MAX                  := "SensorsSettings".AIR1_Max,
           OUT                      := "A_Sensors".AIR1,
           ERROR                    := #xError);
NETWORK
TITLE =
      CALL  "LinTrafo" (
           IN_WORD                  := PIW 314,
           IN_MIN                   := 0.000000e+00,
           IN_MAX                   := 2.764000e+04,
           OUT_MIN                  := "SensorsSettings".QIRAH4H4_Min,
           OUT_MAX                  := "SensorsSettings".QIRAH4H4_Max,
           OUT                      := "A_Sensors".Qirahq4,
           ERROR                    := #xError);
NETWORK
TITLE =
      A     "DI".DI_XL1_QL3;
      =     "_DI_XL1_QL3";
      A     "DI".DI_XL2_QL3;
      =     "_DI_XL2_QL3";
      A     "DI".DI_Q3_Bad;
      =     "_DI_Q3_Bad";
      A     "DI".DI_AB1_Working;
      =     "_DI_AB1_Working";
      A     "DI".DI_Kb_1_1_Working;
      =     "_DI_Kb_1_1_Working";
      A     "DI".DI_Kb_1_1_Alm;
      =     "_DI_Kb_1_1_Alm";
      A     "DI".DI_Kb_1_2_Working;
      =     "_DI_Kb_1_2_Working";
      A     "DI".DI_Kb_1_2_Alm;
      =     "_DI_Kb_1_2_Alm";
      A     "DI".DI_Kb_2_Working;
      =     "_DI_Kb_2_Working";
      A     "DI".DI_Kb_2_Alm;
      =     "_DI_Kb_2_Alm";
      A     "DI".DI_Kd_1_Working;
      =     "_DI_Kd_1_Working";
      A     "DI".DI_Kd_1_Alm;
      =     "_DI_Kd_1_Alm";
      A     "DI".DI_ZB_1_Opn;
      =     "_DI_ZB_1_Opn";
      A     "DI".DI_ZB_1_Cls;
      =     "_DI_ZB_1_Cls";
      A     "DI".DI_ZB_1_Local;
      =     "_DI_ZB_1_Local";
      A     "DI".DI_ZB_1_Alm;
      =     "_DI_ZB_1_Alm";
      A     "DI".DI_ZB_2_Opn;
      =     "_DI_ZB_2_Opn";
      A     "DI".DI_ZB_2_Cls;
      =     "_DI_ZB_2_Cls";
      A     "DI".DI_ZB_2_Local;
      =     "_DI_ZB_2_Local";
      A     "DI".DI_ZB_2_Alm;
      =     "_DI_ZB_2_Alm";
      A     "DI".DI_ZB_3_Opn;
      =     "_DI_ZB_3_Opn";
      A     "DI".DI_ZB_3_Cls;
      =     "_DI_ZB_3_Cls";
      A     "DI".DI_ZB_3_Local;
      =     "_DI_ZB_3_Local";
      A     "DI".DI_ZB_3_Alm;
      =     "_DI_ZB_3_Alm";
      A     "DI".DI_EUV_001_Opn;
      =     "_DI_EUV_001_Opn";
      A     "DI".DI_EUV_001_Cls;
      =     "_DI_EUV_001_Cls";
      A     "DI".DI_EUV_001_Local;
      =     "_DI_EUV_001_Local";
      A     "DI".DI_EUV_001_Alm;
      =     "_DI_EUV_002_Opn";
      A     "DI".DI_EUV_002_Opn;
      =     "_DI_EUV_002_Cls";
      A     "DI".DI_EUV_002_Cls;
      =     "_DI_EUV_002_Local";
      A     "DI".DI_EUV_002_Local;
      =     "_DI_EUV_002_Alm";
      A     "DI".DI_EUV_002_Alm;
      =     "_DI_EUV_003_Opn";
      A     "DI".DI_EUV_003_Opn;
      =     "_DI_EUV_003_Cls";
      A     "DI".DI_EUV_003_Cls;
      =     "_DI_EUV_003_Local";
      A     "DI".DI_EUV_003_Local;
      =     "_DI_EUV_003_Alm";
      A     "DI".DI_EUV_003_Alm;
      =     "QSA_19_1_1";
      A     "DI".DI_KD_1_QSA_1_5QSL1_5_2;
      =     "QSA_23_1_1";
      A     "DI".DI_Q3_BAD_1;
      =     "QSA_19_1_2";
      A     "DI".DI_AB1_XLA_AV1_Alm;
      =     "QSA_23_1_2";
      A     "DI".DI_AB2_XL_AV2_Working;
      =     "QSA_19_1_3";
      A     "DI".DI_AB2_XLA_AV2_Alm;
      =     "QSA_23_1_3";
      A     "DI".DI_AB3_XL_AV3_Working;
      =     "QSA_19_1_4";
      A     "DI".DI_AB3_XLA_AV3_Alm;
      =     "QSA_23_1_4";
      A     "DI".DI_AB4_XL_AV4_Working;
      =     "QSA_19_1_5";
      A     "DI".DI_AB4_XLA_AV4_Alm;
      =     "QSA_23_1_5";
      A     "DI".DI_P2_XLP_2_Working;
      =     "Q3_BAD";
      A     "DI".DI_P2_XLP_2_Alm;
      =     "AB_1_Alm";
      A     "DI".DI_P3_XLP_3_Working;
      =     "AB_2_Working";
      A     "DI".DI_P3_XLP_3_Alm;
      =     "AB_2_Alm";
      A     "DI".DI_IBP_1_Working;
      =     "AB_3_Working";
      A     "DI".DI_IBP_1_Alm;
      =     "AB_3_Alm";
      A     "DI".DI_IBP_1_Bypass;
      =     "AB_4_Working";
      A     "DI".DI_IBP_2_Working;
      =     "AB_4_Alm";
      A     "DI".DI_IBP_2_Alm;
      =     "P2_Alm";
      A     "DI".DI_IBP_2_Bypass;
      =     "P2_Working";
      CALL  "ByteToByte" (
           bIn                      := PIB 0,
           OUT                      := "DI_Bytes".B_0);
      CALL  "ByteToByte" (
           bIn                      := PIB 1,
           OUT                      := "DI_Bytes".B_1);
      CALL  "ByteToByte" (
           bIn                      := PIB 2,
           OUT                      := "DI_Bytes".B_2);
      CALL  "ByteToByte" (
           bIn                      := PIB 3,
           OUT                      := "DI_Bytes".B_3);
      CALL  "ByteToByte" (
           bIn                      := PIB 4,
           OUT                      := "DI_Bytes".B_4);
      CALL  "ByteToByte" (
           bIn                      := PIB 5,
           OUT                      := "DI_Bytes".B_5);
      CALL  "ByteToByte" (
           bIn                      := PIB 6,
           OUT                      := "DI_Bytes".B_6);
      CALL  "ByteToByte" (
           bIn                      := PIB 7,
           OUT                      := "DI_Bytes".B_7);
      CALL  "ByteToByte" (
           bIn                      := PIB 8,
           OUT                      := "DI_Bytes".B_8);
      CALL  "ByteToByte" (
           bIn                      := PIB 9,
           OUT                      := "DI_Bytes".B_9);
      CALL  "ByteToByte" (
           bIn                      := PIB 10,
           OUT                      := "DI_Bytes".B_10);
      CALL  "ByteToByte" (
           bIn                      := PIB 11,
           OUT                      := "DI_Bytes".B_11);
END_FUNCTION_BLOCK

FUNCTION_BLOCK "PO2_GetReals"	// FB 31
VERSION : 0.1
BEGIN
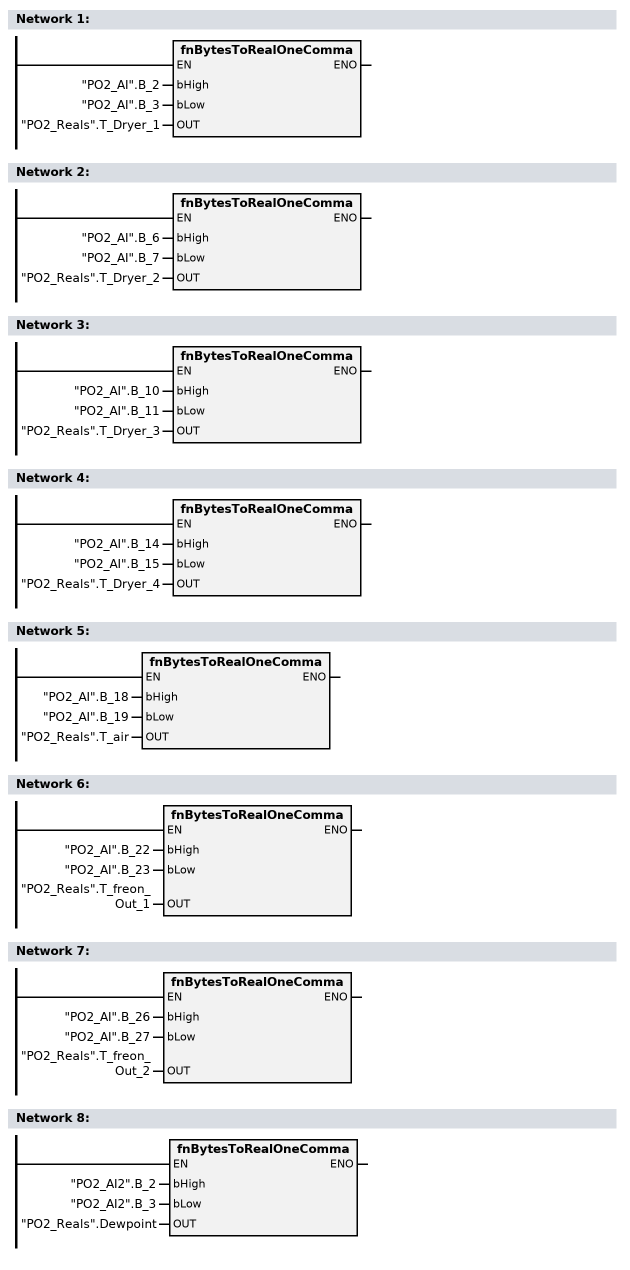
NETWORK
TITLE =
      CALL  "fnBytesToRealOneComma" (
           bHigh                    := "PO2_AI".B_2,
           bLow                     := "PO2_AI".B_3,
           OUT                      := "PO2_Reals".T_Dryer_1);
      NOP   0;
NETWORK
TITLE =
      CALL  "fnBytesToRealOneComma" (
           bHigh                    := "PO2_AI".B_6,
           bLow                     := "PO2_AI".B_7,
           OUT                      := "PO2_Reals".T_Dryer_2);
      NOP   0;
NETWORK
TITLE =
      CALL  "fnBytesToRealOneComma" (
           bHigh                    := "PO2_AI".B_10,
           bLow                     := "PO2_AI".B_11,
           OUT                      := "PO2_Reals".T_Dryer_3);
      NOP   0;
NETWORK
TITLE =
      CALL  "fnBytesToRealOneComma" (
           bHigh                    := "PO2_AI".B_14,
           bLow                     := "PO2_AI".B_15,
           OUT                      := "PO2_Reals".T_Dryer_4);
      NOP   0;
NETWORK
TITLE =
      CALL  "fnBytesToRealOneComma" (
           bHigh                    := "PO2_AI".B_18,
           bLow                     := "PO2_AI".B_19,
           OUT                      := "PO2_Reals".T_air);
      NOP   0;
NETWORK
TITLE =
      CALL  "fnBytesToRealOneComma" (
           bHigh                    := "PO2_AI".B_22,
           bLow                     := "PO2_AI".B_23,
           OUT                      := "PO2_Reals".T_freon_Out_1);
      NOP   0;
NETWORK
TITLE =
      CALL  "fnBytesToRealOneComma" (
           bHigh                    := "PO2_AI".B_26,
           bLow                     := "PO2_AI".B_27,
           OUT                      := "PO2_Reals".T_freon_Out_2);
      NOP   0;
NETWORK
TITLE =
      CALL  "fnBytesToRealOneComma" (
           bHigh                    := "PO2_AI2".B_2,
           bLow                     := "PO2_AI2".B_3,
           OUT                      := "PO2_Reals".Dewpoint);
      NOP   0;
END_FUNCTION_BLOCK

FUNCTION_BLOCK "DI_ToVars"	// FB 32
VERSION : 0.1
VAR_TEMP
  xFalse : BOOL ;
  rCheck : REAL ;
END_VAR
BEGIN
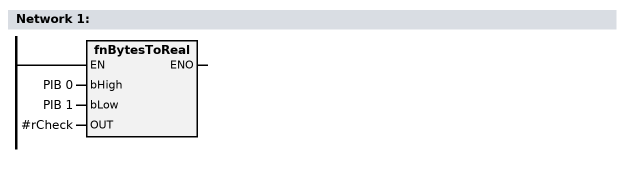
NETWORK
TITLE =
      CALL  "fnBytesToReal" (
           bHigh                    := PIB 0,
           bLow                     := PIB 1,
           OUT                      := #rCheck);
      NOP   0;
NETWORK
TITLE =
END_FUNCTION_BLOCK

FUNCTION_BLOCK "Valve_PID"	// FB 33
VERSION : 0.1
VAR_INPUT
  rSetPressure : REAL ;
  xManual : BOOL ;
  rSetManualPercent : REAL ;
  rKp : REAL  := 5.000000e+000;
  tKi : TIME  := T#3M20S;
  tKd : TIME ;
  rFeedback : REAL ;
END_VAR
VAR_OUTPUT
  rOut : REAL ;
  wOutAO : WORD ;
END_VAR
BEGIN
